(* CODESYS project barrier.v1.12.paramReset.project

Project tree, tasks and I/O mapping:
  Device : ShenZhen RenTong SoftMotion RTE V3,  Shenzhen Rentong IST LTD, order no. 309015, version 3.5.9.50
    application Application
      libraries: Standard, * (System); VisuDialogs, * (System); SysDir, 3.5.8.0 (System); SysTime23, 3.5.2.0 (System); TCP, 3.5.9.50 (3S - Smart Software Solutions GmbH); SysFile, 3.5.9.0 (System); SysStr23, 3.5.8.0 (System); modbus tcp serverAndClient, 1.0.1 (深圳人通长沙研究院); ModbusTCP Slave, 3.5.10.0 (3S - Smart Software Solutions GmbH)
      task CAN_TX (cyclic, interval t#10ms, priority 1) calls CanTx
      task CAN_RX (cyclic, interval 6 ms, priority 1) calls CanRx
      task MAIN (cyclic, interval t#10ms, priority 2) calls Barrier
      task VISU_TASK (cyclic, interval 100 ms, priority 31) calls VisuElems.Visu_Prg
      task MODBUS (cyclic, interval t#10ms, priority 1) calls ModbusAct
      task ETHERCAT (cyclic, interval 2000 µs, priority 0) calls EtherCAT_Master.EtherCAT_Task [EtherCAT_Master.EtherCAT_Task]
      task HEALTHY_DATA1 (cyclic, interval t#500ms, priority 1) calls TcpUploader
      task HEALTHY_DATA2 (cyclic, interval t#10ms, priority 1) calls FileSaver
      basestruct/
        data type CmdPercentSet
        data type SensorInfo
        data type DeviceUnit
        data type UIMode
        data type UIUnit
        data type TargetDirect
        data type DevStatus
      can/
        canstruct/
          data type Can_BUS_8Inputs
          data type Can_BUS_8Outputs
          data type Can_Bus_RXMsg_Buff
          data type Can_Bus_TXMsg_Buff
          data type Can_baseframe
        program CanTx [ST]: C01_Tx, C02_Tx, C03_Tx, C04_Tx, C05_Tx, C06_Tx
        program CanRx [ST]: C01_Rx, C02_Rx, C03_Rx, C04_Rx, C05_Rx, C06_Rx
        function CAN_Read_Data_SWMC [ST]
        function CAN_Send_Data_SWMC [ST]
      global/
        global variables gController
        global variables gCan
        global variables gDev
        global variables gUI
        global variables gModbus
      visualization/
        baseModule/
          visualisation DevUnit0
          visualisation grd
          visualisation setting
          visualisation sky
          visualisation BasePID
          visualisation testPID
          visualisation currentUnit
      core/
        program Barrier [ST]: updateStatus, initialize, interfaceAct, autoResetButton, manualExecute, pidExecute, pidTestUi, autoEnable, pidCalc, setExecutePercent, initializePid
        pid/
          function block BasePIDCtrl [ST]
          data type PidParam
          data type UiPid
          data type DevPid
          function block grdPosCtrl [ST]
          function block skyPosCtrl [ST]
          data type FeedForward
      visualisation main
      healthydata/
        program TcpUploader [ST]: prepareMetaData
        program FileSaver [ST]: getSkyData, getGrdData
      modbus/
        struct/
          data type mdbsStruct
          data type mdbsRequest
          data type mdbsResponse
        program ModbusAct [ST]: initialize, localCmdHandler, updateStat, handleCmd, handleStat1, handleStat2, handleStat3, localStatHandler
        function block mdbsLogicToPhy [ST]
        function block mdbsPhyToLogic [ST]
        function block mdbsNumToIdx [ST]
        function block DataReverse [ST]: cmdReverse
      atrace/
        trace delay_g_07 (task MAIN, trigger Positive on CanRx.count 1): gController.grd[7].retractPercent, gController.grd[7].extendPercent, gDev.grd[7].sensor.position, gDev.grd[7].sensor.speed
        trace show (task MAIN, trigger Positive on CanRx.count 1): gDev.grd[9].sensor.position, gDev.grd[9].sensor.speed, Barrier.grdPid[9].res, gController.grd[9].retractPercent, gController.grd[9].extendPercent, gDev.sky[9].sensor.position, gDev.sky[9].sensor.speed, Barrier.skyPid[9].res, gController.sky[9].retractPercent, gController.sky[9].extendPercent
        trace delay_g_08 (task MAIN, trigger Positive on CanRx.count 1): gController.grd[8].retractPercent, gController.grd[8].extendPercent, gDev.grd[8].sensor.position, gDev.grd[8].sensor.speed
        trace show2 (task MAIN, trigger Positive on CanRx.count 1): gController.grd[1].retractPercent, gController.grd[1].extendPercent, gDev.grd[1].sensor.position, gDev.grd[1].sensor.speed
        sync/
          trace delay_sync_01 (task MAIN, trigger Positive on CanRx.count 1): gDev.grd[1].sensor.position, gDev.grd[1].sensor.speed, gDev.sky[1].sensor.position, gDev.sky[1].sensor.speed
          trace delay_sync_02 (task MAIN, trigger Positive on CanRx.count 1): gDev.grd[2].sensor.position, gDev.grd[2].sensor.speed, gDev.sky[2].sensor.position, gDev.sky[2].sensor.speed
          trace delay_sync_03 (task MAIN, trigger Positive on CanRx.count 1): gDev.grd[3].sensor.position, gDev.grd[3].sensor.speed, gDev.sky[3].sensor.position, gDev.sky[3].sensor.speed
          trace delay_sync_04 (task MAIN, trigger Positive on CanRx.count 1): gDev.grd[4].sensor.position, gDev.grd[4].sensor.speed, gDev.sky[4].sensor.position, gDev.sky[4].sensor.speed
          trace delay_sync_05 (task MAIN, trigger Positive on CanRx.count 1): gDev.grd[5].sensor.position, gDev.grd[5].sensor.speed, gDev.sky[5].sensor.position, gDev.sky[5].sensor.speed
          trace delay_sync_06 (task MAIN, trigger Positive on CanRx.count 1): gDev.grd[6].sensor.position, gDev.grd[6].sensor.speed, gDev.sky[6].sensor.position, gDev.sky[6].sensor.speed
          trace delay_sync_07 (task MAIN, trigger Positive on CanRx.count 1): gDev.grd[7].sensor.position, gDev.grd[7].sensor.speed, gDev.sky[7].sensor.position, gDev.sky[7].sensor.speed
          trace delay_sync_08 (task MAIN, trigger Positive on CanRx.count 1): gDev.grd[8].sensor.position, gDev.grd[8].sensor.speed, gDev.sky[8].sensor.position, gDev.sky[8].sensor.speed
          trace delay_sync_09 (task MAIN, trigger Positive on CanRx.count 1): gDev.grd[9].sensor.position, gDev.grd[9].sensor.speed, gDev.sky[9].sensor.position, gDev.sky[9].sensor.speed
          trace delay_sync_10 (task MAIN, trigger Positive on CanRx.count 1): gDev.grd[10].sensor.position, gDev.grd[10].sensor.speed, gDev.sky[10].sensor.position, gDev.sky[10].sensor.speed
        last/
          trace delay_s_0 (task MAIN, trigger Positive on CanRx.count 1): gController.sky[0].retractPercent, gController.sky[0].extendPercent, gDev.sky[0].sensor.position, gDev.sky[0].sensor.speed
          trace delay_g_5 (task MAIN, trigger Positive on CanRx.count 1): gController.grd[5].retractPercent, gController.grd[5].extendPercent, gDev.grd[5].sensor.position, gDev.grd[5].sensor.speed
          trace delay_g_1 (task MAIN, trigger Positive on CanRx.count 1): gController.grd[1].retractPercent, gController.grd[1].extendPercent, gDev.grd[1].sensor.position, gDev.grd[1].sensor.speed
          trace delay_g_2 (task MAIN, trigger Positive on CanRx.count 1): gController.grd[2].retractPercent, gController.grd[2].extendPercent, gDev.grd[2].sensor.position, gDev.grd[2].sensor.speed
          trace delay_g_3 (task MAIN, trigger Positive on CanRx.count 1): gController.grd[3].retractPercent, gController.grd[3].extendPercent, gDev.grd[3].current[1], gDev.grd[3].current[2], gDev.grd[3].sensor.position, gDev.grd[3].sensor.speed
          trace delay_g_4 (task MAIN, trigger Positive on CanRx.count 1): gController.grd[4].retractPercent, gController.grd[4].extendPercent, gDev.grd[4].current[1], gDev.grd[4].current[2], gDev.grd[4].sensor.position, gDev.grd[4].sensor.speed
          trace delay_g_6 (task MAIN, trigger Positive on CanRx.count 1): gController.grd[6].retractPercent, gController.grd[6].extendPercent, gDev.grd[6].current[1], gDev.grd[6].current[2], gDev.grd[6].sensor.position, gDev.grd[6].sensor.speed
          trace delay_s_6 (task MAIN, trigger Positive on CanRx.count 1): gController.sky[6].retractPercent, gController.sky[6].extendPercent, gDev.sky[6].sensor.position, gDev.sky[6].sensor.speed
          trace delay_s_5 (task MAIN, trigger Positive on CanRx.count 1): gController.sky[5].retractPercent, gController.sky[5].extendPercent, gDev.sky[5].sensor.position, gDev.sky[5].sensor.speed
          trace delay_s_4 (task MAIN, trigger Positive on CanRx.count 1): gController.sky[4].retractPercent, gController.sky[4].extendPercent, gDev.sky[4].sensor.position, gDev.sky[4].sensor.speed
          trace delay_s_3 (task MAIN, trigger Positive on CanRx.count 1): gController.sky[3].retractPercent, gController.sky[3].extendPercent, gDev.sky[3].sensor.position, gDev.sky[3].sensor.speed
          trace delay_s_2 (task MAIN, trigger Positive on CanRx.count 1): gController.sky[2].retractPercent, gController.sky[2].extendPercent, gDev.sky[2].sensor.position, gDev.sky[2].sensor.speed
          trace delay_s_1 (task MAIN, trigger Positive on CanRx.count 1): gController.sky[1].retractPercent, gController.sky[1].extendPercent, gDev.sky[1].sensor.position, gDev.sky[1].sensor.speed
        trace delay_g_09 (task MAIN, trigger Positive on CanRx.count 1): gController.grd[9].retractPercent, gController.grd[9].extendPercent, gDev.grd[9].sensor.position, gDev.grd[9].sensor.speed
        trace delay_g_10 (task MAIN, trigger Positive on CanRx.count 1): gController.grd[10].retractPercent, gController.grd[10].extendPercent, gDev.grd[10].sensor.position, gDev.grd[10].sensor.speed
        trace delay_s_07 (task MAIN, trigger Positive on CanRx.count 1): gController.sky[07].retractPercent, gController.sky[07].extendPercent, gDev.sky[07].sensor.position, gDev.sky[07].sensor.speed
        trace delay_s_08 (task MAIN, trigger Positive on CanRx.count 1): gController.sky[8].retractPercent, gController.sky[8].extendPercent, gDev.sky[8].sensor.position, gDev.sky[8].sensor.speed
        trace delay_s_09 (task MAIN, trigger Positive on CanRx.count 1): gDev.grd[9].sensor.position, gDev.grd[9].sensor.speed, Barrier.grdPid[9].res, gController.grd[9].retractPercent, gController.grd[9].extendPercent, gDev.sky[9].sensor.position, gDev.sky[9].sensor.speed, Barrier.skyPid[9].res, gController.sky[9].retractPercent, gController.sky[9].extendPercent
        trace delay_s_10 (task MAIN, trigger Positive on CanRx.count 1): gController.sky[10].retractPercent, gController.sky[10].extendPercent, gDev.sky[10].sensor.position, gDev.sky[10].sensor.speed
      basefun/
        function block CommandExecutor0 [ST]
        function percentCalc [ST]
        function setButtonByDirect [ST]
        function updateDevStatus [ST]
        function block tcpUpload [ST]: send
        function block fileSave [ST]: new, close, write, createDir
        function block CommandExecutor [ST]
    SoftMotion General Axis Pool
    EtherCAT_Master : EtherCAT Master, 3S - Smart Software Solutions GmbH, version 3.5.10.0
        settings: MasterCycleTime = 2000; NetworkName = '本地连接 5'; NetworkName = "本地连接 5"; SrcAddress1 = 26861; SrcAddress2 = 2754393510
      EK1100_0030 : EK1100-0030 EtherCAT Coupler (2A E-Bus, 4kV galv. iso.), Beckhoff Automation GmbH & Co. KG, order no. EK1100-0030, version Revision=16#0011001E
          settings: DC sync0 cycletime = 2000; DC sync1 cycletime = 2000
        EL6751_CANMiniDriver : EL6751 CAN MiniDriver (8 Messages), Beckhoff Automation GmbH, version 3.5.9.0
            settings: DC sync0 cycletime = 2000; DC sync1 cycletime = 2000
            unmapped channels: TxCounter, RxCounter, NoOfTxMessages, TxMsg1_TransactionNumber, TxMsg1_CobId, TxMsg1_Byte1, TxMsg1_Byte2, TxMsg1_Byte3, TxMsg1_Byte4, TxMsg1_Byte5, TxMsg1_Byte6, TxMsg1_Byte7, TxMsg1_Byte8, TxMsg2_TransactionNumber, TxMsg2_CobId, TxMsg2_Byte1, TxMsg2_Byte2, TxMsg2_Byte3, TxMsg2_Byte4, TxMsg2_Byte5, TxMsg2_Byte6, TxMsg2_Byte7, TxMsg2_Byte8, TxMsg3_TransactionNumber, TxMsg3_CobId, TxMsg3_Byte1, TxMsg3_Byte2, TxMsg3_Byte3, TxMsg3_Byte4, TxMsg3_Byte5, TxMsg3_Byte6, TxMsg3_Byte7, TxMsg3_Byte8, TxMsg4_TransactionNumber, TxMsg4_CobId, TxMsg4_Byte1, TxMsg4_Byte2, TxMsg4_Byte3, TxMsg4_Byte4, TxMsg4_Byte5,
              TxMsg4_Byte6, TxMsg4_Byte7, TxMsg4_Byte8, TxMsg5_TransactionNumber, TxMsg5_CobId, TxMsg5_Byte1, TxMsg5_Byte2, TxMsg5_Byte3, TxMsg5_Byte4, TxMsg5_Byte5, TxMsg5_Byte6, TxMsg5_Byte7, TxMsg5_Byte8, TxMsg6_TransactionNumber, TxMsg6_CobId, TxMsg6_Byte1, TxMsg6_Byte2, TxMsg6_Byte3, TxMsg6_Byte4, TxMsg6_Byte5, TxMsg6_Byte6, TxMsg6_Byte7, TxMsg6_Byte8, TxMsg7_TransactionNumber, TxMsg7_CobId, TxMsg7_Byte1, TxMsg7_Byte2, TxMsg7_Byte3, TxMsg7_Byte4, TxMsg7_Byte5, TxMsg7_Byte6, TxMsg7_Byte7, TxMsg7_Byte8, TxMsg8_TransactionNumber, TxMsg8_CobId, TxMsg8_Byte1, TxMsg8_Byte2, TxMsg8_Byte3, TxMsg8_Byte4, TxMsg8_Byte5,
              TxMsg8_Byte6, TxMsg8_Byte7, TxMsg8_Byte8, CAN Control, TxCounter, RxCounter, NoOfRxMessages, TransactionNumber, RxMsg1_CobId, RxMsg1_Byte1, RxMsg1_Byte2, RxMsg1_Byte3, RxMsg1_Byte4, RxMsg1_Byte5, RxMsg1_Byte6, RxMsg1_Byte7, RxMsg1_Byte8, RxMsg2_CobId, RxMsg2_Byte1, RxMsg2_Byte2, RxMsg2_Byte3, RxMsg2_Byte4, RxMsg2_Byte5, RxMsg2_Byte6, RxMsg2_Byte7, RxMsg2_Byte8, RxMsg3_CobId, RxMsg3_Byte1, RxMsg3_Byte2, RxMsg3_Byte3, RxMsg3_Byte4, RxMsg3_Byte5, RxMsg3_Byte6, RxMsg3_Byte7, RxMsg3_Byte8, RxMsg4_CobId, RxMsg4_Byte1, RxMsg4_Byte2, RxMsg4_Byte3, RxMsg4_Byte4,
              RxMsg4_Byte5, RxMsg4_Byte6, RxMsg4_Byte7, RxMsg4_Byte8, RxMsg5_CobId, RxMsg5_Byte1, RxMsg5_Byte2, RxMsg5_Byte3, RxMsg5_Byte4, RxMsg5_Byte5, RxMsg5_Byte6, RxMsg5_Byte7, RxMsg5_Byte8, RxMsg6_CobId, RxMsg6_Byte1, RxMsg6_Byte2, RxMsg6_Byte3, RxMsg6_Byte4, RxMsg6_Byte5, RxMsg6_Byte6, RxMsg6_Byte7, RxMsg6_Byte8, RxMsg7_CobId, RxMsg7_Byte1, RxMsg7_Byte2, RxMsg7_Byte3, RxMsg7_Byte4, RxMsg7_Byte5, RxMsg7_Byte6, RxMsg7_Byte7, RxMsg7_Byte8, RxMsg8_CobId, RxMsg8_Byte1, RxMsg8_Byte2, RxMsg8_Byte3, RxMsg8_Byte4, RxMsg8_Byte5, RxMsg8_Byte6, RxMsg8_Byte7, RxMsg8_Byte8,
              CAN State, Align, RX Error Counter, TX Error Counter
          CANbus
      EK1100_0030_1 : EK1100-0030 EtherCAT Coupler (2A E-Bus, 4kV galv. iso.), Beckhoff Automation GmbH & Co. KG, order no. EK1100-0030, version Revision=16#0011001E
          settings: DC sync0 cycletime = 2000; DC sync1 cycletime = 2000
        EL6751_CANMiniDriver_1 : EL6751 CAN MiniDriver (8 Messages), Beckhoff Automation GmbH, version 3.5.9.0
            settings: DC sync0 cycletime = 2000; DC sync1 cycletime = 2000
            unmapped channels: TxCounter, RxCounter, NoOfTxMessages, TxMsg1_TransactionNumber, TxMsg1_CobId, TxMsg1_Byte1, TxMsg1_Byte2, TxMsg1_Byte3, TxMsg1_Byte4, TxMsg1_Byte5, TxMsg1_Byte6, TxMsg1_Byte7, TxMsg1_Byte8, TxMsg2_TransactionNumber, TxMsg2_CobId, TxMsg2_Byte1, TxMsg2_Byte2, TxMsg2_Byte3, TxMsg2_Byte4, TxMsg2_Byte5, TxMsg2_Byte6, TxMsg2_Byte7, TxMsg2_Byte8, TxMsg3_TransactionNumber, TxMsg3_CobId, TxMsg3_Byte1, TxMsg3_Byte2, TxMsg3_Byte3, TxMsg3_Byte4, TxMsg3_Byte5, TxMsg3_Byte6, TxMsg3_Byte7, TxMsg3_Byte8, TxMsg4_TransactionNumber, TxMsg4_CobId, TxMsg4_Byte1, TxMsg4_Byte2, TxMsg4_Byte3, TxMsg4_Byte4, TxMsg4_Byte5,
              TxMsg4_Byte6, TxMsg4_Byte7, TxMsg4_Byte8, TxMsg5_TransactionNumber, TxMsg5_CobId, TxMsg5_Byte1, TxMsg5_Byte2, TxMsg5_Byte3, TxMsg5_Byte4, TxMsg5_Byte5, TxMsg5_Byte6, TxMsg5_Byte7, TxMsg5_Byte8, TxMsg6_TransactionNumber, TxMsg6_CobId, TxMsg6_Byte1, TxMsg6_Byte2, TxMsg6_Byte3, TxMsg6_Byte4, TxMsg6_Byte5, TxMsg6_Byte6, TxMsg6_Byte7, TxMsg6_Byte8, TxMsg7_TransactionNumber, TxMsg7_CobId, TxMsg7_Byte1, TxMsg7_Byte2, TxMsg7_Byte3, TxMsg7_Byte4, TxMsg7_Byte5, TxMsg7_Byte6, TxMsg7_Byte7, TxMsg7_Byte8, TxMsg8_TransactionNumber, TxMsg8_CobId, TxMsg8_Byte1, TxMsg8_Byte2, TxMsg8_Byte3, TxMsg8_Byte4, TxMsg8_Byte5,
              TxMsg8_Byte6, TxMsg8_Byte7, TxMsg8_Byte8, CAN Control, TxCounter, RxCounter, NoOfRxMessages, TransactionNumber, RxMsg1_CobId, RxMsg1_Byte1, RxMsg1_Byte2, RxMsg1_Byte3, RxMsg1_Byte4, RxMsg1_Byte5, RxMsg1_Byte6, RxMsg1_Byte7, RxMsg1_Byte8, RxMsg2_CobId, RxMsg2_Byte1, RxMsg2_Byte2, RxMsg2_Byte3, RxMsg2_Byte4, RxMsg2_Byte5, RxMsg2_Byte6, RxMsg2_Byte7, RxMsg2_Byte8, RxMsg3_CobId, RxMsg3_Byte1, RxMsg3_Byte2, RxMsg3_Byte3, RxMsg3_Byte4, RxMsg3_Byte5, RxMsg3_Byte6, RxMsg3_Byte7, RxMsg3_Byte8, RxMsg4_CobId, RxMsg4_Byte1, RxMsg4_Byte2, RxMsg4_Byte3, RxMsg4_Byte4,
              RxMsg4_Byte5, RxMsg4_Byte6, RxMsg4_Byte7, RxMsg4_Byte8, RxMsg5_CobId, RxMsg5_Byte1, RxMsg5_Byte2, RxMsg5_Byte3, RxMsg5_Byte4, RxMsg5_Byte5, RxMsg5_Byte6, RxMsg5_Byte7, RxMsg5_Byte8, RxMsg6_CobId, RxMsg6_Byte1, RxMsg6_Byte2, RxMsg6_Byte3, RxMsg6_Byte4, RxMsg6_Byte5, RxMsg6_Byte6, RxMsg6_Byte7, RxMsg6_Byte8, RxMsg7_CobId, RxMsg7_Byte1, RxMsg7_Byte2, RxMsg7_Byte3, RxMsg7_Byte4, RxMsg7_Byte5, RxMsg7_Byte6, RxMsg7_Byte7, RxMsg7_Byte8, RxMsg8_CobId, RxMsg8_Byte1, RxMsg8_Byte2, RxMsg8_Byte3, RxMsg8_Byte4, RxMsg8_Byte5, RxMsg8_Byte6, RxMsg8_Byte7, RxMsg8_Byte8,
              CAN State, Align, RX Error Counter, TX Error Counter
          CANbus
              settings: NetID = 1
      EK1100_0030_2 : EK1100-0030 EtherCAT Coupler (2A E-Bus, 4kV galv. iso.), Beckhoff Automation GmbH & Co. KG, order no. EK1100-0030, version Revision=16#0011001E
          settings: DC sync0 cycletime = 2000; DC sync1 cycletime = 2000
        EL6751_CANMiniDriver_2 : EL6751 CAN MiniDriver (8 Messages), Beckhoff Automation GmbH, version 3.5.9.0
            settings: DC sync0 cycletime = 2000; DC sync1 cycletime = 2000
            unmapped channels: TxCounter, RxCounter, NoOfTxMessages, TxMsg1_TransactionNumber, TxMsg1_CobId, TxMsg1_Byte1, TxMsg1_Byte2, TxMsg1_Byte3, TxMsg1_Byte4, TxMsg1_Byte5, TxMsg1_Byte6, TxMsg1_Byte7, TxMsg1_Byte8, TxMsg2_TransactionNumber, TxMsg2_CobId, TxMsg2_Byte1, TxMsg2_Byte2, TxMsg2_Byte3, TxMsg2_Byte4, TxMsg2_Byte5, TxMsg2_Byte6, TxMsg2_Byte7, TxMsg2_Byte8, TxMsg3_TransactionNumber, TxMsg3_CobId, TxMsg3_Byte1, TxMsg3_Byte2, TxMsg3_Byte3, TxMsg3_Byte4, TxMsg3_Byte5, TxMsg3_Byte6, TxMsg3_Byte7, TxMsg3_Byte8, TxMsg4_TransactionNumber, TxMsg4_CobId, TxMsg4_Byte1, TxMsg4_Byte2, TxMsg4_Byte3, TxMsg4_Byte4, TxMsg4_Byte5,
              TxMsg4_Byte6, TxMsg4_Byte7, TxMsg4_Byte8, TxMsg5_TransactionNumber, TxMsg5_CobId, TxMsg5_Byte1, TxMsg5_Byte2, TxMsg5_Byte3, TxMsg5_Byte4, TxMsg5_Byte5, TxMsg5_Byte6, TxMsg5_Byte7, TxMsg5_Byte8, TxMsg6_TransactionNumber, TxMsg6_CobId, TxMsg6_Byte1, TxMsg6_Byte2, TxMsg6_Byte3, TxMsg6_Byte4, TxMsg6_Byte5, TxMsg6_Byte6, TxMsg6_Byte7, TxMsg6_Byte8, TxMsg7_TransactionNumber, TxMsg7_CobId, TxMsg7_Byte1, TxMsg7_Byte2, TxMsg7_Byte3, TxMsg7_Byte4, TxMsg7_Byte5, TxMsg7_Byte6, TxMsg7_Byte7, TxMsg7_Byte8, TxMsg8_TransactionNumber, TxMsg8_CobId, TxMsg8_Byte1, TxMsg8_Byte2, TxMsg8_Byte3, TxMsg8_Byte4, TxMsg8_Byte5,
              TxMsg8_Byte6, TxMsg8_Byte7, TxMsg8_Byte8, CAN Control, TxCounter, RxCounter, NoOfRxMessages, TransactionNumber, RxMsg1_CobId, RxMsg1_Byte1, RxMsg1_Byte2, RxMsg1_Byte3, RxMsg1_Byte4, RxMsg1_Byte5, RxMsg1_Byte6, RxMsg1_Byte7, RxMsg1_Byte8, RxMsg2_CobId, RxMsg2_Byte1, RxMsg2_Byte2, RxMsg2_Byte3, RxMsg2_Byte4, RxMsg2_Byte5, RxMsg2_Byte6, RxMsg2_Byte7, RxMsg2_Byte8, RxMsg3_CobId, RxMsg3_Byte1, RxMsg3_Byte2, RxMsg3_Byte3, RxMsg3_Byte4, RxMsg3_Byte5, RxMsg3_Byte6, RxMsg3_Byte7, RxMsg3_Byte8, RxMsg4_CobId, RxMsg4_Byte1, RxMsg4_Byte2, RxMsg4_Byte3, RxMsg4_Byte4,
              RxMsg4_Byte5, RxMsg4_Byte6, RxMsg4_Byte7, RxMsg4_Byte8, RxMsg5_CobId, RxMsg5_Byte1, RxMsg5_Byte2, RxMsg5_Byte3, RxMsg5_Byte4, RxMsg5_Byte5, RxMsg5_Byte6, RxMsg5_Byte7, RxMsg5_Byte8, RxMsg6_CobId, RxMsg6_Byte1, RxMsg6_Byte2, RxMsg6_Byte3, RxMsg6_Byte4, RxMsg6_Byte5, RxMsg6_Byte6, RxMsg6_Byte7, RxMsg6_Byte8, RxMsg7_CobId, RxMsg7_Byte1, RxMsg7_Byte2, RxMsg7_Byte3, RxMsg7_Byte4, RxMsg7_Byte5, RxMsg7_Byte6, RxMsg7_Byte7, RxMsg7_Byte8, RxMsg8_CobId, RxMsg8_Byte1, RxMsg8_Byte2, RxMsg8_Byte3, RxMsg8_Byte4, RxMsg8_Byte5, RxMsg8_Byte6, RxMsg8_Byte7, RxMsg8_Byte8,
              CAN State, Align, RX Error Counter, TX Error Counter
          CANbus
              settings: NetID = 2
      EK1100_0030_3 : EK1100-0030 EtherCAT Coupler (2A E-Bus, 4kV galv. iso.), Beckhoff Automation GmbH & Co. KG, order no. EK1100-0030, version Revision=16#0011001E
          settings: DC sync0 cycletime = 2000; DC sync1 cycletime = 2000
        EL6751_CANMiniDriver_3 : EL6751 CAN MiniDriver (8 Messages), Beckhoff Automation GmbH, version 3.5.9.0
            settings: DC sync0 cycletime = 2000; DC sync1 cycletime = 2000
            unmapped channels: TxCounter, RxCounter, NoOfTxMessages, TxMsg1_TransactionNumber, TxMsg1_CobId, TxMsg1_Byte1, TxMsg1_Byte2, TxMsg1_Byte3, TxMsg1_Byte4, TxMsg1_Byte5, TxMsg1_Byte6, TxMsg1_Byte7, TxMsg1_Byte8, TxMsg2_TransactionNumber, TxMsg2_CobId, TxMsg2_Byte1, TxMsg2_Byte2, TxMsg2_Byte3, TxMsg2_Byte4, TxMsg2_Byte5, TxMsg2_Byte6, TxMsg2_Byte7, TxMsg2_Byte8, TxMsg3_TransactionNumber, TxMsg3_CobId, TxMsg3_Byte1, TxMsg3_Byte2, TxMsg3_Byte3, TxMsg3_Byte4, TxMsg3_Byte5, TxMsg3_Byte6, TxMsg3_Byte7, TxMsg3_Byte8, TxMsg4_TransactionNumber, TxMsg4_CobId, TxMsg4_Byte1, TxMsg4_Byte2, TxMsg4_Byte3, TxMsg4_Byte4, TxMsg4_Byte5,
              TxMsg4_Byte6, TxMsg4_Byte7, TxMsg4_Byte8, TxMsg5_TransactionNumber, TxMsg5_CobId, TxMsg5_Byte1, TxMsg5_Byte2, TxMsg5_Byte3, TxMsg5_Byte4, TxMsg5_Byte5, TxMsg5_Byte6, TxMsg5_Byte7, TxMsg5_Byte8, TxMsg6_TransactionNumber, TxMsg6_CobId, TxMsg6_Byte1, TxMsg6_Byte2, TxMsg6_Byte3, TxMsg6_Byte4, TxMsg6_Byte5, TxMsg6_Byte6, TxMsg6_Byte7, TxMsg6_Byte8, TxMsg7_TransactionNumber, TxMsg7_CobId, TxMsg7_Byte1, TxMsg7_Byte2, TxMsg7_Byte3, TxMsg7_Byte4, TxMsg7_Byte5, TxMsg7_Byte6, TxMsg7_Byte7, TxMsg7_Byte8, TxMsg8_TransactionNumber, TxMsg8_CobId, TxMsg8_Byte1, TxMsg8_Byte2, TxMsg8_Byte3, TxMsg8_Byte4, TxMsg8_Byte5,
              TxMsg8_Byte6, TxMsg8_Byte7, TxMsg8_Byte8, CAN Control, TxCounter, RxCounter, NoOfRxMessages, TransactionNumber, RxMsg1_CobId, RxMsg1_Byte1, RxMsg1_Byte2, RxMsg1_Byte3, RxMsg1_Byte4, RxMsg1_Byte5, RxMsg1_Byte6, RxMsg1_Byte7, RxMsg1_Byte8, RxMsg2_CobId, RxMsg2_Byte1, RxMsg2_Byte2, RxMsg2_Byte3, RxMsg2_Byte4, RxMsg2_Byte5, RxMsg2_Byte6, RxMsg2_Byte7, RxMsg2_Byte8, RxMsg3_CobId, RxMsg3_Byte1, RxMsg3_Byte2, RxMsg3_Byte3, RxMsg3_Byte4, RxMsg3_Byte5, RxMsg3_Byte6, RxMsg3_Byte7, RxMsg3_Byte8, RxMsg4_CobId, RxMsg4_Byte1, RxMsg4_Byte2, RxMsg4_Byte3, RxMsg4_Byte4,
              RxMsg4_Byte5, RxMsg4_Byte6, RxMsg4_Byte7, RxMsg4_Byte8, RxMsg5_CobId, RxMsg5_Byte1, RxMsg5_Byte2, RxMsg5_Byte3, RxMsg5_Byte4, RxMsg5_Byte5, RxMsg5_Byte6, RxMsg5_Byte7, RxMsg5_Byte8, RxMsg6_CobId, RxMsg6_Byte1, RxMsg6_Byte2, RxMsg6_Byte3, RxMsg6_Byte4, RxMsg6_Byte5, RxMsg6_Byte6, RxMsg6_Byte7, RxMsg6_Byte8, RxMsg7_CobId, RxMsg7_Byte1, RxMsg7_Byte2, RxMsg7_Byte3, RxMsg7_Byte4, RxMsg7_Byte5, RxMsg7_Byte6, RxMsg7_Byte7, RxMsg7_Byte8, RxMsg8_CobId, RxMsg8_Byte1, RxMsg8_Byte2, RxMsg8_Byte3, RxMsg8_Byte4, RxMsg8_Byte5, RxMsg8_Byte6, RxMsg8_Byte7, RxMsg8_Byte8,
              CAN State, Align, RX Error Counter, TX Error Counter
          CANbus
              settings: NetID = 3
      EK1100_0030_4 : EK1100-0030 EtherCAT Coupler (2A E-Bus, 4kV galv. iso.), Beckhoff Automation GmbH & Co. KG, order no. EK1100-0030, version Revision=16#0011001E
          settings: DC sync0 cycletime = 2000; DC sync1 cycletime = 2000
        EL6751_CANMiniDriver_4 : EL6751 CAN MiniDriver (8 Messages), Beckhoff Automation GmbH, version 3.5.9.0
            settings: DC sync0 cycletime = 2000; DC sync1 cycletime = 2000
            unmapped channels: TxCounter, RxCounter, NoOfTxMessages, TxMsg1_TransactionNumber, TxMsg1_CobId, TxMsg1_Byte1, TxMsg1_Byte2, TxMsg1_Byte3, TxMsg1_Byte4, TxMsg1_Byte5, TxMsg1_Byte6, TxMsg1_Byte7, TxMsg1_Byte8, TxMsg2_TransactionNumber, TxMsg2_CobId, TxMsg2_Byte1, TxMsg2_Byte2, TxMsg2_Byte3, TxMsg2_Byte4, TxMsg2_Byte5, TxMsg2_Byte6, TxMsg2_Byte7, TxMsg2_Byte8, TxMsg3_TransactionNumber, TxMsg3_CobId, TxMsg3_Byte1, TxMsg3_Byte2, TxMsg3_Byte3, TxMsg3_Byte4, TxMsg3_Byte5, TxMsg3_Byte6, TxMsg3_Byte7, TxMsg3_Byte8, TxMsg4_TransactionNumber, TxMsg4_CobId, TxMsg4_Byte1, TxMsg4_Byte2, TxMsg4_Byte3, TxMsg4_Byte4, TxMsg4_Byte5,
              TxMsg4_Byte6, TxMsg4_Byte7, TxMsg4_Byte8, TxMsg5_TransactionNumber, TxMsg5_CobId, TxMsg5_Byte1, TxMsg5_Byte2, TxMsg5_Byte3, TxMsg5_Byte4, TxMsg5_Byte5, TxMsg5_Byte6, TxMsg5_Byte7, TxMsg5_Byte8, TxMsg6_TransactionNumber, TxMsg6_CobId, TxMsg6_Byte1, TxMsg6_Byte2, TxMsg6_Byte3, TxMsg6_Byte4, TxMsg6_Byte5, TxMsg6_Byte6, TxMsg6_Byte7, TxMsg6_Byte8, TxMsg7_TransactionNumber, TxMsg7_CobId, TxMsg7_Byte1, TxMsg7_Byte2, TxMsg7_Byte3, TxMsg7_Byte4, TxMsg7_Byte5, TxMsg7_Byte6, TxMsg7_Byte7, TxMsg7_Byte8, TxMsg8_TransactionNumber, TxMsg8_CobId, TxMsg8_Byte1, TxMsg8_Byte2, TxMsg8_Byte3, TxMsg8_Byte4, TxMsg8_Byte5,
              TxMsg8_Byte6, TxMsg8_Byte7, TxMsg8_Byte8, CAN Control, TxCounter, RxCounter, NoOfRxMessages, TransactionNumber, RxMsg1_CobId, RxMsg1_Byte1, RxMsg1_Byte2, RxMsg1_Byte3, RxMsg1_Byte4, RxMsg1_Byte5, RxMsg1_Byte6, RxMsg1_Byte7, RxMsg1_Byte8, RxMsg2_CobId, RxMsg2_Byte1, RxMsg2_Byte2, RxMsg2_Byte3, RxMsg2_Byte4, RxMsg2_Byte5, RxMsg2_Byte6, RxMsg2_Byte7, RxMsg2_Byte8, RxMsg3_CobId, RxMsg3_Byte1, RxMsg3_Byte2, RxMsg3_Byte3, RxMsg3_Byte4, RxMsg3_Byte5, RxMsg3_Byte6, RxMsg3_Byte7, RxMsg3_Byte8, RxMsg4_CobId, RxMsg4_Byte1, RxMsg4_Byte2, RxMsg4_Byte3, RxMsg4_Byte4,
              RxMsg4_Byte5, RxMsg4_Byte6, RxMsg4_Byte7, RxMsg4_Byte8, RxMsg5_CobId, RxMsg5_Byte1, RxMsg5_Byte2, RxMsg5_Byte3, RxMsg5_Byte4, RxMsg5_Byte5, RxMsg5_Byte6, RxMsg5_Byte7, RxMsg5_Byte8, RxMsg6_CobId, RxMsg6_Byte1, RxMsg6_Byte2, RxMsg6_Byte3, RxMsg6_Byte4, RxMsg6_Byte5, RxMsg6_Byte6, RxMsg6_Byte7, RxMsg6_Byte8, RxMsg7_CobId, RxMsg7_Byte1, RxMsg7_Byte2, RxMsg7_Byte3, RxMsg7_Byte4, RxMsg7_Byte5, RxMsg7_Byte6, RxMsg7_Byte7, RxMsg7_Byte8, RxMsg8_CobId, RxMsg8_Byte1, RxMsg8_Byte2, RxMsg8_Byte3, RxMsg8_Byte4, RxMsg8_Byte5, RxMsg8_Byte6, RxMsg8_Byte7, RxMsg8_Byte8,
              CAN State, Align, RX Error Counter, TX Error Counter
          CANbus
              settings: NetID = 4
      EK1100_0030_5 : EK1100-0030 EtherCAT Coupler (2A E-Bus, 4kV galv. iso.), Beckhoff Automation GmbH & Co. KG, order no. EK1100-0030, version Revision=16#0011001E
          settings: DC sync0 cycletime = 2000; DC sync1 cycletime = 2000
        EL6751_CANMiniDriver_5 : EL6751 CAN MiniDriver (8 Messages), Beckhoff Automation GmbH, version 3.5.9.0
            settings: DC sync0 cycletime = 2000; DC sync1 cycletime = 2000
            unmapped channels: TxCounter, RxCounter, NoOfTxMessages, TxMsg1_TransactionNumber, TxMsg1_CobId, TxMsg1_Byte1, TxMsg1_Byte2, TxMsg1_Byte3, TxMsg1_Byte4, TxMsg1_Byte5, TxMsg1_Byte6, TxMsg1_Byte7, TxMsg1_Byte8, TxMsg2_TransactionNumber, TxMsg2_CobId, TxMsg2_Byte1, TxMsg2_Byte2, TxMsg2_Byte3, TxMsg2_Byte4, TxMsg2_Byte5, TxMsg2_Byte6, TxMsg2_Byte7, TxMsg2_Byte8, TxMsg3_TransactionNumber, TxMsg3_CobId, TxMsg3_Byte1, TxMsg3_Byte2, TxMsg3_Byte3, TxMsg3_Byte4, TxMsg3_Byte5, TxMsg3_Byte6, TxMsg3_Byte7, TxMsg3_Byte8, TxMsg4_TransactionNumber, TxMsg4_CobId, TxMsg4_Byte1, TxMsg4_Byte2, TxMsg4_Byte3, TxMsg4_Byte4, TxMsg4_Byte5,
              TxMsg4_Byte6, TxMsg4_Byte7, TxMsg4_Byte8, TxMsg5_TransactionNumber, TxMsg5_CobId, TxMsg5_Byte1, TxMsg5_Byte2, TxMsg5_Byte3, TxMsg5_Byte4, TxMsg5_Byte5, TxMsg5_Byte6, TxMsg5_Byte7, TxMsg5_Byte8, TxMsg6_TransactionNumber, TxMsg6_CobId, TxMsg6_Byte1, TxMsg6_Byte2, TxMsg6_Byte3, TxMsg6_Byte4, TxMsg6_Byte5, TxMsg6_Byte6, TxMsg6_Byte7, TxMsg6_Byte8, TxMsg7_TransactionNumber, TxMsg7_CobId, TxMsg7_Byte1, TxMsg7_Byte2, TxMsg7_Byte3, TxMsg7_Byte4, TxMsg7_Byte5, TxMsg7_Byte6, TxMsg7_Byte7, TxMsg7_Byte8, TxMsg8_TransactionNumber, TxMsg8_CobId, TxMsg8_Byte1, TxMsg8_Byte2, TxMsg8_Byte3, TxMsg8_Byte4, TxMsg8_Byte5,
              TxMsg8_Byte6, TxMsg8_Byte7, TxMsg8_Byte8, CAN Control, TxCounter, RxCounter, NoOfRxMessages, TransactionNumber, RxMsg1_CobId, RxMsg1_Byte1, RxMsg1_Byte2, RxMsg1_Byte3, RxMsg1_Byte4, RxMsg1_Byte5, RxMsg1_Byte6, RxMsg1_Byte7, RxMsg1_Byte8, RxMsg2_CobId, RxMsg2_Byte1, RxMsg2_Byte2, RxMsg2_Byte3, RxMsg2_Byte4, RxMsg2_Byte5, RxMsg2_Byte6, RxMsg2_Byte7, RxMsg2_Byte8, RxMsg3_CobId, RxMsg3_Byte1, RxMsg3_Byte2, RxMsg3_Byte3, RxMsg3_Byte4, RxMsg3_Byte5, RxMsg3_Byte6, RxMsg3_Byte7, RxMsg3_Byte8, RxMsg4_CobId, RxMsg4_Byte1, RxMsg4_Byte2, RxMsg4_Byte3, RxMsg4_Byte4,
              RxMsg4_Byte5, RxMsg4_Byte6, RxMsg4_Byte7, RxMsg4_Byte8, RxMsg5_CobId, RxMsg5_Byte1, RxMsg5_Byte2, RxMsg5_Byte3, RxMsg5_Byte4, RxMsg5_Byte5, RxMsg5_Byte6, RxMsg5_Byte7, RxMsg5_Byte8, RxMsg6_CobId, RxMsg6_Byte1, RxMsg6_Byte2, RxMsg6_Byte3, RxMsg6_Byte4, RxMsg6_Byte5, RxMsg6_Byte6, RxMsg6_Byte7, RxMsg6_Byte8, RxMsg7_CobId, RxMsg7_Byte1, RxMsg7_Byte2, RxMsg7_Byte3, RxMsg7_Byte4, RxMsg7_Byte5, RxMsg7_Byte6, RxMsg7_Byte7, RxMsg7_Byte8, RxMsg8_CobId, RxMsg8_Byte1, RxMsg8_Byte2, RxMsg8_Byte3, RxMsg8_Byte4, RxMsg8_Byte5, RxMsg8_Byte6, RxMsg8_Byte7, RxMsg8_Byte8,
              CAN State, Align, RX Error Counter, TX Error Counter
          CANbus
              settings: NetID = 5
  libraries: VisuSymbols, 3.5.10.0 (System)
  text list GlobalTextList
*)

// Device/Application/can/canstruct/Can_BUS_8Inputs
TYPE Can_BUS_8Inputs :          //输入缓存结构 EL2721-8Message_IN
STRUCT
	TxCounter			: UINT;
	RxCounter			: UINT;
	NoOfRxMessages 	 	: UINT;
	TransactionNumber	: UINT;
	RXMsg				: ARRAY[1..8] OF Can_Bus_RXMsg_Buff;
	CAN_State			: UINT;
	Align				: UINT;
	RX_Error_Cnt		: BYTE;
	TX_Error_Cnt		: BYTE;
END_STRUCT
END_TYPE

// Device/Application/can/canstruct/Can_BUS_8Outputs
TYPE Can_BUS_8Outputs :		//输出缓存结构 EL2721-8Message_OUT
STRUCT
	TxCounter		: UINT;
	RxCounter		: UINT;
	NoOfTxMessages 	: UINT;
	TXMsg			: ARRAY[1..8] OF Can_Bus_TXMsg_Buff;
	CAN_Control		: UINT;
END_STRUCT
END_TYPE

// Device/Application/can/canstruct/Can_Bus_RXMsg_Buff
TYPE Can_Bus_RXMsg_Buff:
STRUCT
	RxMsg_CobId		: UINT;
	RxMsg_Byte  	: ARRAY[1..8] OF BYTE;
END_STRUCT
END_TYPE

// Device/Application/can/canstruct/Can_Bus_TXMsg_Buff
TYPE Can_Bus_TXMsg_Buff :
STRUCT
	TxMsg_TransactionNumber		: UINT;
	TxMsg_CobId					: UINT;
	TxMsg_Byte  				: ARRAY[1..8] OF BYTE;
END_STRUCT
END_TYPE

// Device/Application/can/canstruct/Can_baseframe
TYPE Can_baseframe :
STRUCT
	id		: UINT;
	data	: ARRAY[1..8] OF BYTE;
END_STRUCT
END_TYPE

// Device/Application/basestruct/CmdPercentSet
TYPE CmdPercentSet :
STRUCT
	extendPercent		:WORD;		//0-65535
	retractPercent		:WORD;		//0-65535
END_STRUCT
END_TYPE

// Device/Application/basestruct/SensorInfo
TYPE SensorInfo :
STRUCT
	
	position	:REAL;	//实时位移
	speed		:REAL;	//实时速度
	
	//记录最大最小位移值
	retractVal	:REAL;	//缩回到位值
	extendVal	:REAL;	//伸出到位值
	
END_STRUCT
END_TYPE

// Device/Application/basestruct/DeviceUnit
TYPE DeviceUnit :
STRUCT
		
	sensor			:SensorInfo;		//传感器参数
	ctrl			:DevPid;			//pid等计算控制执行参数	
	
	vector			:TargetDirect;		//指令运行方向 1-伸出 2-缩回 3-停止
	state			:DevStatus;			//设备状态 0-未知 1-运行 2-伸出到位 3-缩回到位 4-错误
	
	timeCounter		:INT;				//timeoutCounter超时计数器
	exeCounter		:INT;				//ExecuteCounter额外执行时间计数

	current			:ARRAY[1..2] OF WORD;	//电流mA	[i,j] -> 地轨挡板i的电流，j=1伸出电流，j=2缩回电流


END_STRUCT
END_TYPE

// Device/Application/basestruct/UIMode
TYPE UIMode :
STRUCT
	manualButtonSet			:BOOL;		//手动复位按钮模式
	usePID					:BOOL;		//使用pid
	autoEnable				:BOOL;		//自动使能
	manualPercentSet		:BOOL;		//手动设定比例量
	manualSetPid			:BOOL;		//手动调节pid参数，可通过pid测试界面设定目标位移值
	
	syncExt					:BOOL;		//同步伸
	syncRct					:BOOL;		//同步缩
	
	hydPowerOn				:BOOL;		//液压站开启 modbus 使用
	hydPowerOff				:BOOL;		//液压站关闭 modbus 使用
	hydPowerReset			:BOOL;		
END_STRUCT
END_TYPE

// Device/Application/basestruct/UIUnit
TYPE UIUnit :
STRUCT
	//cmd
	pwrEnable			:BOOL;		//比例阀使能   power-enable
	pwrPercent			:REAL;		//比例阀百分比 power-percent 0-100
	
	//button
	btnExtend			:BOOL;
	btnRetract			:BOOL;
	btnStop				:BOOL;
	btnLast				:TargetDirect;	//上次动作方向
	
	//info display
	name				:STRING;	//挡板名
	wname				:WSTRING;	//山河命名
	hzname				:WSTRING;	//hua zhong ming ming
	postion				:REAL;		//位移值
	speed				:REAL;
	extendPercent		:REAL;		//伸出百分比 extend-percent
	
	
	
END_STRUCT
END_TYPE

// Device/Application/basestruct/TargetDirect
{attribute 'qualified_only'}
{attribute 'strict'}
TYPE TargetDirect :
(
	extend 	:= 1,	//伸出
	
	retract := 2,	//缩回
	
	stop	:= 3	//停止
);
END_TYPE

// Device/Application/basestruct/DevStatus
{attribute 'qualified_only'}
{attribute 'strict'}
TYPE DevStatus :
(
	unknown 	:= 0,
	
	runing		:= 1,
	
	extended	:= 2,
	
	retracted	:= 3,
	
	error		:= 4
);
END_TYPE

// Device/Application/core/pid/PidParam
TYPE PidParam :
STRUCT
	Kp			:REAL;
	Ki			:REAL;
	Kd			:REAL;
	Set_Point	:REAL;
	Max_Val		:REAL;
	Max_ACC		:REAL;
	Act_Val		:REAL;
	Err			:REAL;
	OUT			:REAL;
END_STRUCT
END_TYPE

// Device/Application/core/pid/UiPid
TYPE UiPid :
STRUCT
	pos				:PidParam;			//位置pid参数
	spd				:PidParam;			//速度pid参数
	ff				:FeedForward;		//前馈参数

	level			:INT;				//1->地轨	2->天轨
	idx				:INT;				//挡板索引编号
	
	devSetPos		:REAL;				//设备中的设定位置点(用于观测)
	executeVal		:REAL;				//执行值(-100.0~+100.0)

	
	posBtn			:BOOL;			//位置控制按钮，按下实时更新交互参数
	rstPidBtn		:BOOL;			//reset pid param button重置pid参数按钮
	pwrPercent		:REAL;			//比例阀百分比 power-percent 0-100	
	
	
	
	
	extendBtn		:BOOL;
	retractBtn		:BOOL;
	stopBtn			:BOOL;


	
	
(*	posErr			:REAL;
	posOut			:REAL;
	spdErr			:REAL;
	spdOut			:REAL;*)	
END_STRUCT
END_TYPE

// Device/Application/core/pid/DevPid
TYPE DevPid :
STRUCT
	pos			:PidParam;			//位置pid参数
	spd			:PidParam;			//速度pid参数
	ff			:FeedForward;		//前馈参数
//	dp			:DynamicPlanning;	//规划参数
	exPct		:REAL;				//伸出默认比例量0-100
	rtPct		:REAL;				//缩回默认比例量0-100
	
	isError		:BOOL;				//当传感器数据为0时，报错并不执行pid
	
	extVal		:REAL;				//设定伸出位移值
	rtcVal		:REAL;				//设定缩回位移值
	
END_STRUCT
END_TYPE

// Device/Application/modbus/struct/mdbsStruct
TYPE mdbsStruct :
STRUCT
	request		:mdbsRequest;				//请求动作指令
	response	:mdbsResponse;			//响应动作指令-天地轨所有	
	
END_STRUCT
END_TYPE

// Device/Application/modbus/struct/mdbsRequest
TYPE mdbsRequest :	//所有请求动作指令数据
STRUCT
	startAddr		:WORD;					//解析起始地址->10
	length			:WORD;					//数据长度/字节->48
	data			:ARRAY[10..57] OF WORD;	//指令数据	
	
	arrNew		:ARRAY [1..4,0..15] OF BOOL;
	arrLast		:ARRAY [1..4,0..15] OF BOOL;

END_STRUCT
END_TYPE

// Device/Application/modbus/struct/mdbsResponse
TYPE mdbsResponse :	//所有响应状态数据回送
STRUCT
	startAddr		:WORD;							//解析起始地址->110
	length			:WORD;							//字节长度->210
	
	data			:ARRAY[110..319] OF WORD;		//位置数据

END_STRUCT
END_TYPE

// Device/Application/core/pid/FeedForward
TYPE FeedForward :
STRUCT
	
	pstThreshold	:REAL;	//正向设定阈值	
	pstKv			:REAL;
	pstKa			:REAL;
	pstKaa			:REAL;
	negThreshold	:REAL;	//反向设定阈值
	negKv			:REAL;
	negKa			:REAL;
	negKaa			:REAL;
	

	
//	pstFactor		:REAL;	//正向设定速度系数因子
//	negFactor		:REAL;	//反向设定速度系数因子


END_STRUCT
END_TYPE

// Device/Application/global/gController
{attribute 'qualified_only'}
VAR_GLOBAL
	//发送至SWMC的比例阀的控制指令
	sky		:ARRAY[0..10] OF CmdPercentSet;
	grd		:ARRAY[1..10] OF CmdPercentSet;
END_VAR

// Device/Application/global/gCan
{attribute 'qualified_only'}
VAR_GLOBAL
	C6TxMsg			AT%QW00		:Can_BUS_8Outputs;	
	C6RxMsg			AT%IW00		:Can_BUS_8Inputs;
	C6RxCounter			 	   	:UINT;
	
	C3TxMsg			AT%QW52		:Can_BUS_8Outputs;	
	C3RxMsg			AT%IW47		:Can_BUS_8Inputs;
	C3RxCounter			   	   	:UINT;

	C4TxMsg			AT%QW104	:Can_BUS_8Outputs;	
	C4RxMsg			AT%IW94		:Can_BUS_8Inputs;
	C4RxCounter				  	:UINT;

	C2TxMsg			AT%QW156	:Can_BUS_8Outputs;	
	C2RxMsg			AT%IW141	:Can_BUS_8Inputs;
	C2RxCounter			 	   	:UINT;
//(*	
	C1TxMsg			AT%QW208	:Can_BUS_8Outputs;	
	C1RxMsg			AT%IW188	:Can_BUS_8Inputs;
	C1RxCounter			   	   	:UINT;

	C5TxMsg			AT%QW260	:Can_BUS_8Outputs;	
	C5RxMsg			AT%IW235	:Can_BUS_8Inputs;
	C5RxCounter				  	:UINT;
//*)

END_VAR

// Device/Application/global/gDev
{attribute 'qualified_only'}
VAR_GLOBAL
	sky		:ARRAY[0..10] OF DeviceUnit;
	grd		:ARRAY[1..10] OF DeviceUnit;
END_VAR

// Device/Application/global/gUI
{attribute 'qualified_only'}
VAR_GLOBAL
	
	mode	:UIMode;					//模式设定

	sky		:ARRAY[0..10] OF UIUnit;	//挡板2组
	grd		:ARRAY[1..10] OF UIUnit;	//挡板1组
	
	pid		:UiPid;						//pid测试界面参数
	
	
	
END_VAR

// Device/Application/global/gModbus
{attribute 'qualified_only'}
VAR_GLOBAL CONSTANT
	g_modbusDataSizeMax	:  UINT:=65535; // 从机保持寄存器数量
END_VAR
VAR_GLOBAL
	srv				:mdbsStruct;		//modbus-service
	modbusBuffer	:ARRAY[0..g_modbusDataSizeMax] OF WORD;	//输入寄存器数据区	
END_VAR

// Device/Application/can/CanTx
PROGRAM CanTx
VAR
	count		:UINT;
END_VAR

count := count + 1;
IF count > 1000 THEN
	count := 1;
END_IF

C01_Tx();
C02_Tx();
C03_Tx();
C04_Tx();
C05_Tx();
C06_Tx();

METHOD C01_Tx
VAR_INPUT
END_VAR
VAR
	swmcIdSwtich		:UINT;
	sendData			:ARRAY[1..8] OF BYTE;
END_VAR

swmcIdSwtich := count MOD 2;
CASE swmcIdSwtich OF
	0:
		sendData[1] := WORD_TO_BYTE(gController.sky[3].extendPercent);
		sendData[2] := WORD_TO_BYTE(SHR(gController.sky[3].extendPercent,8));
		sendData[3] := WORD_TO_BYTE(gController.sky[3].retractPercent);
		sendData[4] := WORD_TO_BYTE(SHR(gController.sky[3].retractPercent,8));
		sendData[5] := WORD_TO_BYTE(gController.sky[4].extendPercent);
		sendData[6] := WORD_TO_BYTE(SHR(gController.sky[4].extendPercent,8));
		sendData[7] := WORD_TO_BYTE(gController.sky[4].retractPercent);
		sendData[8] := WORD_TO_BYTE(SHR(gController.sky[4].retractPercent,8));
		CAN_Send_Data_SWMC(1, 16#500,senddata);   //发送ID 0x460到C6
		
	1:
		sendData[1] := WORD_TO_BYTE(gController.sky[5].extendPercent);
		sendData[2] := WORD_TO_BYTE(SHR(gController.sky[5].extendPercent,8));
		sendData[3] := WORD_TO_BYTE(gController.sky[5].retractPercent);
		sendData[4] := WORD_TO_BYTE(SHR(gController.sky[5].retractPercent,8));
		sendData[5] := WORD_TO_BYTE(gController.sky[6].extendPercent);
		sendData[6] := WORD_TO_BYTE(SHR(gController.sky[6].extendPercent,8));
		sendData[7] := WORD_TO_BYTE(gController.sky[6].retractPercent);
		sendData[8] := WORD_TO_BYTE(SHR(gController.sky[6].retractPercent,8));
		CAN_Send_Data_SWMC(1, 16#501,senddata);   //发送ID 0x460到C6
		
		


END_CASE
END_METHOD

METHOD C02_Tx
VAR_INPUT
END_VAR
VAR
	swmcIdSwtich		:UINT;
	sendData			:ARRAY[1..8] OF BYTE;
END_VAR

swmcIdSwtich := count MOD 2;
CASE swmcIdSwtich OF
	0:
		sendData[1] := WORD_TO_BYTE(gController.sky[0].extendPercent);
		sendData[2] := WORD_TO_BYTE(SHR(gController.sky[0].extendPercent,8));
		sendData[3] := WORD_TO_BYTE(gController.sky[0].retractPercent);
		sendData[4] := WORD_TO_BYTE(SHR(gController.sky[0].retractPercent,8));
		sendData[5] := WORD_TO_BYTE(gController.sky[1].extendPercent);
		sendData[6] := WORD_TO_BYTE(SHR(gController.sky[1].extendPercent,8));
		sendData[7] := WORD_TO_BYTE(gController.sky[1].retractPercent);
		sendData[8] := WORD_TO_BYTE(SHR(gController.sky[1].retractPercent,8));
		CAN_Send_Data_SWMC(2, 16#510,senddata);   //发送ID 0x460到C6
		
	1:
		sendData[1] := WORD_TO_BYTE(gController.sky[2].extendPercent);
		sendData[2] := WORD_TO_BYTE(SHR(gController.sky[2].extendPercent,8));
		sendData[3] := WORD_TO_BYTE(gController.sky[2].retractPercent);
		sendData[4] := WORD_TO_BYTE(SHR(gController.sky[2].retractPercent,8));
		CAN_Send_Data_SWMC(2, 16#511,senddata);   //发送ID 0x460到C6
		
		


END_CASE
END_METHOD

METHOD C03_Tx
VAR_INPUT
END_VAR
VAR
	swmcIdSwtich		:UINT;
	sendData			:ARRAY[1..8] OF BYTE;
END_VAR

swmcIdSwtich := count MOD 2;
CASE swmcIdSwtich OF
	0:
		sendData[1] := WORD_TO_BYTE(gController.grd[3].extendPercent);
		sendData[2] := WORD_TO_BYTE(SHR(gController.grd[3].extendPercent,8));
		sendData[3] := WORD_TO_BYTE(gController.grd[3].retractPercent);
		sendData[4] := WORD_TO_BYTE(SHR(gController.grd[3].retractPercent,8));
		sendData[5] := WORD_TO_BYTE(gController.grd[4].extendPercent);
		sendData[6] := WORD_TO_BYTE(SHR(gController.grd[4].extendPercent,8));
		sendData[7] := WORD_TO_BYTE(gController.grd[4].retractPercent);
		sendData[8] := WORD_TO_BYTE(SHR(gController.grd[4].retractPercent,8));
		CAN_Send_Data_SWMC(3, 16#520,senddata);   //发送ID 0x460到C6
		
	1:
		sendData[1] := WORD_TO_BYTE(gController.grd[5].extendPercent);
		sendData[2] := WORD_TO_BYTE(SHR(gController.grd[5].extendPercent,8));
		sendData[3] := WORD_TO_BYTE(gController.grd[5].retractPercent);
		sendData[4] := WORD_TO_BYTE(SHR(gController.grd[5].retractPercent,8));
		sendData[5] := WORD_TO_BYTE(gController.grd[6].extendPercent);
		sendData[6] := WORD_TO_BYTE(SHR(gController.grd[6].extendPercent,8));
		sendData[7] := WORD_TO_BYTE(gController.grd[6].retractPercent);
		sendData[8] := WORD_TO_BYTE(SHR(gController.grd[6].retractPercent,8));
		CAN_Send_Data_SWMC(3, 16#521,senddata);   //发送ID 0x460到C6
		
		


END_CASE
END_METHOD

METHOD C04_Tx
VAR_INPUT
END_VAR
VAR
	swmcIdSwtich		:UINT;
	sendData			:ARRAY[1..8] OF BYTE;
END_VAR

swmcIdSwtich := count MOD 2;
CASE swmcIdSwtich OF
	0:
		sendData[1] := WORD_TO_BYTE(gController.grd[1].extendPercent);
		sendData[2] := WORD_TO_BYTE(SHR(gController.grd[1].extendPercent,8));
		sendData[3] := WORD_TO_BYTE(gController.grd[1].retractPercent);
		sendData[4] := WORD_TO_BYTE(SHR(gController.grd[1].retractPercent,8));
		sendData[5] := WORD_TO_BYTE(gController.grd[2].extendPercent);
		sendData[6] := WORD_TO_BYTE(SHR(gController.grd[2].extendPercent,8));
		sendData[7] := WORD_TO_BYTE(gController.grd[2].retractPercent);
		sendData[8] := WORD_TO_BYTE(SHR(gController.grd[2].retractPercent,8));
		CAN_Send_Data_SWMC(4, 16#530,senddata);   //发送ID 0x460到C6
		
		
		


END_CASE
END_METHOD

METHOD C05_Tx
VAR_INPUT
END_VAR
VAR
	swmcIdSwtich		:UINT;
	sendData			:ARRAY[1..8] OF BYTE;
END_VAR

swmcIdSwtich := count MOD 2;
CASE swmcIdSwtich OF
	0:
		sendData[1] := WORD_TO_BYTE(gController.sky[7].extendPercent);
		sendData[2] := WORD_TO_BYTE(SHR(gController.sky[7].extendPercent,8));
		sendData[3] := WORD_TO_BYTE(gController.sky[7].retractPercent);
		sendData[4] := WORD_TO_BYTE(SHR(gController.sky[7].retractPercent,8));
		sendData[5] := WORD_TO_BYTE(gController.sky[8].extendPercent);
		sendData[6] := WORD_TO_BYTE(SHR(gController.sky[8].extendPercent,8));
		sendData[7] := WORD_TO_BYTE(gController.sky[8].retractPercent);
		sendData[8] := WORD_TO_BYTE(SHR(gController.sky[8].retractPercent,8));
		CAN_Send_Data_SWMC(5, 16#540,senddata);   //发送ID 0x460到C6	
	1:
		sendData[1] := WORD_TO_BYTE(gController.sky[9].extendPercent);
		sendData[2] := WORD_TO_BYTE(SHR(gController.sky[9].extendPercent,8));
		sendData[3] := WORD_TO_BYTE(gController.sky[9].retractPercent);
		sendData[4] := WORD_TO_BYTE(SHR(gController.sky[9].retractPercent,8));
		sendData[5] := WORD_TO_BYTE(gController.sky[10].extendPercent);
		sendData[6] := WORD_TO_BYTE(SHR(gController.sky[10].extendPercent,8));
		sendData[7] := WORD_TO_BYTE(gController.sky[10].retractPercent);
		sendData[8] := WORD_TO_BYTE(SHR(gController.sky[10].retractPercent,8));
		CAN_Send_Data_SWMC(5, 16#541,senddata);   //发送ID 0x460到C6		

END_CASE
END_METHOD

METHOD C06_Tx
VAR_INPUT
END_VAR
VAR
	swmcIdSwtich		:UINT;
	sendData			:ARRAY[1..8] OF BYTE;
END_VAR

swmcIdSwtich := count MOD 2;
CASE swmcIdSwtich OF
	0:
		sendData[1] := WORD_TO_BYTE(gController.grd[7].extendPercent);
		sendData[2] := WORD_TO_BYTE(SHR(gController.grd[7].extendPercent,8));
		sendData[3] := WORD_TO_BYTE(gController.grd[7].retractPercent);
		sendData[4] := WORD_TO_BYTE(SHR(gController.grd[7].retractPercent,8));
		sendData[5] := WORD_TO_BYTE(gController.grd[8].extendPercent);
		sendData[6] := WORD_TO_BYTE(SHR(gController.grd[8].extendPercent,8));
		sendData[7] := WORD_TO_BYTE(gController.grd[8].retractPercent);
		sendData[8] := WORD_TO_BYTE(SHR(gController.grd[8].retractPercent,8));
		CAN_Send_Data_SWMC(6, 16#550,senddata);   //发送ID 0x460到C6
		
	1:
		sendData[1] := WORD_TO_BYTE(gController.grd[9].extendPercent);
		sendData[2] := WORD_TO_BYTE(SHR(gController.grd[9].extendPercent,8));
		sendData[3] := WORD_TO_BYTE(gController.grd[9].retractPercent);
		sendData[4] := WORD_TO_BYTE(SHR(gController.grd[9].retractPercent,8));
		sendData[5] := WORD_TO_BYTE(gController.grd[10].extendPercent);
		sendData[6] := WORD_TO_BYTE(SHR(gController.grd[10].extendPercent,8));
		sendData[7] := WORD_TO_BYTE(gController.grd[10].retractPercent);
		sendData[8] := WORD_TO_BYTE(SHR(gController.grd[10].retractPercent,8));
		CAN_Send_Data_SWMC(6, 16#551,senddata);   //发送ID 0x460到C6
		
END_CASE
END_METHOD

END_PROGRAM

// Device/Application/can/CAN_Send_Data_SWMC
FUNCTION CAN_Send_Data_SWMC : BOOL
VAR_INPUT
	SWMC_ID : UINT;
	id 		: UINT;
	data	: ARRAY[1..8] OF BYTE;
END_VAR
VAR
	
END_VAR

CASE  SWMC_ID OF

	1:
		gCan.C1TxMsg.TXMsg[1].TxMsg_CobId 	:= 8 + 32 * id;
	  	gCan.C1TxMsg.TXMsg[1].TxMsg_Byte 	:= data;
	   	gCan.C1TxMsg.NoOfTxMessages			:= 1;
	   	gCan.C1TxMsg.TxCounter 				:= gCan.C1TxMsg.TxCounter +1;	
	2:
		gCan.C2TxMsg.TXMsg[1].TxMsg_CobId 	:= 8 + 32 * id;
	  	gCan.C2TxMsg.TXMsg[1].TxMsg_Byte 	:= data;
	   	gCan.C2TxMsg.NoOfTxMessages			:= 1;
	   	gCan.C2TxMsg.TxCounter 				:= gCan.C2TxMsg.TxCounter +1;	
	3:
		gCan.C3TxMsg.TXMsg[1].TxMsg_CobId 	:= 8 + 32 * id;
	  	gCan.C3TxMsg.TXMsg[1].TxMsg_Byte 	:= data;
	   	gCan.C3TxMsg.NoOfTxMessages			:= 1;
	   	gCan.C3TxMsg.TxCounter 				:= gCan.C3TxMsg.TxCounter +1;
	4:
		gCan.C4TxMsg.TXMsg[1].TxMsg_CobId 	:= 8 + 32 * id;
	  	gCan.C4TxMsg.TXMsg[1].TxMsg_Byte 	:= data;
	   	gCan.C4TxMsg.NoOfTxMessages			:= 1;
	   	gCan.C4TxMsg.TxCounter 				:= gCan.C4TxMsg.TxCounter +1;
	//(*
	5:
		gCan.C5TxMsg.TXMsg[1].TxMsg_CobId 	:= 8 + 32 * id;
	  	gCan.C5TxMsg.TXMsg[1].TxMsg_Byte 	:= data;
	   	gCan.C5TxMsg.NoOfTxMessages			:= 1;
	   	gCan.C5TxMsg.TxCounter 				:= gCan.C5TxMsg.TxCounter +1;
	6:
		gCan.C6TxMsg.TXMsg[1].TxMsg_CobId 	:= 8 + 32 * id;
	  	gCan.C6TxMsg.TXMsg[1].TxMsg_Byte 	:= data;
	   	gCan.C6TxMsg.NoOfTxMessages			:= 1;
	   	gCan.C6TxMsg.TxCounter 				:= gCan.C6TxMsg.TxCounter +1;
	//*)

END_CASE

END_FUNCTION

// Device/Application/can/CanRx
PROGRAM CanRx
VAR
	count		:UINT;
END_VAR

count := count + 1;
IF count > 1000 THEN
	count := 1;
END_IF

C01_Rx();
C02_Rx();
C03_Rx();
C04_Rx();
C05_Rx();
C06_Rx();

METHOD C01_Rx
VAR_INPUT
END_VAR
VAR
	frame	 	    :Can_baseframe;
	I				:UINT;
	fId				:UINT;
	pos				:WORD;
	spd				:WORD;
END_VAR
IF gCan.C1RxMsg.RxCounter <>  gCan.C1RxCounter THEN    //接收到新的数据
	FOR I := 1 TO gCan.C1RxMsg.NoOfRxMessages DO
		frame := CAN_Read_Data_SWMC(1,I);
		fId := frame.id;
		CASE fId OF
			16#600:
				pos := BYTE_TO_WORD(frame.data[ 1 ]) OR SHL(BYTE_TO_WORD(frame.data[ 2 ]),8);
				gDev.sky[4].sensor.position := pos * 0.1;
				pos := BYTE_TO_WORD(frame.data[ 3 ]) OR SHL(BYTE_TO_WORD(frame.data[ 4 ]),8);
				gDev.sky[5].sensor.position := pos * 0.1;
				pos := BYTE_TO_WORD(frame.data[ 5 ]) OR SHL(BYTE_TO_WORD(frame.data[ 6 ]),8);
				gDev.sky[6].sensor.position := pos * 0.1;
				pos := BYTE_TO_WORD(frame.data[ 7 ]) OR SHL(BYTE_TO_WORD(frame.data[ 8 ]),8);
				gDev.sky[3].sensor.position := pos * 0.1;
			16#601:
				spd := BYTE_TO_WORD(frame.data[ 1 ]) OR SHL(BYTE_TO_WORD(frame.data[ 2 ]),8);
				gDev.sky[4].sensor.speed := INT_TO_REAL(WORD_TO_INT(spd));
				spd := BYTE_TO_WORD(frame.data[ 3 ]) OR SHL(BYTE_TO_WORD(frame.data[ 4 ]),8);
				gDev.sky[5].sensor.speed := INT_TO_REAL(WORD_TO_INT(spd));
				spd := BYTE_TO_WORD(frame.data[ 5 ]) OR SHL(BYTE_TO_WORD(frame.data[ 6 ]),8);
				gDev.sky[6].sensor.speed := INT_TO_REAL(WORD_TO_INT(spd));
				spd := BYTE_TO_WORD(frame.data[ 7 ]) OR SHL(BYTE_TO_WORD(frame.data[ 8 ]),8);
				gDev.sky[3].sensor.speed := INT_TO_REAL(WORD_TO_INT(spd));
		END_CASE

	END_FOR
	gCan.C1RxCounter := gCan.C1RxMsg.RxCounter;
END_IF
END_METHOD

METHOD C02_Rx
VAR_INPUT
END_VAR
VAR
	frame	 	    :Can_baseframe;
	I				:UINT;
	fId				:UINT;
	pos				:WORD;
	spd				:WORD;
END_VAR
IF gCan.C2RxMsg.RxCounter <>  gCan.C2RxCounter THEN    //接收到新的数据
	FOR I := 1 TO gCan.C2RxMsg.NoOfRxMessages DO
		frame := CAN_Read_Data_SWMC(2,I);
		fId := frame.id;
		CASE fId OF
			16#610:
				pos := BYTE_TO_WORD(frame.data[ 1 ]) OR SHL(BYTE_TO_WORD(frame.data[ 2 ]),8);
				gDev.sky[0].sensor.position := pos * 0.1;
				pos := BYTE_TO_WORD(frame.data[ 3 ]) OR SHL(BYTE_TO_WORD(frame.data[ 4 ]),8);
				gDev.sky[1].sensor.position := pos * 0.1;
				pos := BYTE_TO_WORD(frame.data[ 5 ]) OR SHL(BYTE_TO_WORD(frame.data[ 6 ]),8);
				gDev.sky[2].sensor.position := pos * 0.1;
	
			16#611:
				spd := BYTE_TO_WORD(frame.data[ 1 ]) OR SHL(BYTE_TO_WORD(frame.data[ 2 ]),8);
				gDev.sky[0].sensor.speed := INT_TO_REAL(WORD_TO_INT(spd));
				spd := BYTE_TO_WORD(frame.data[ 3 ]) OR SHL(BYTE_TO_WORD(frame.data[ 4 ]),8);
				gDev.sky[1].sensor.speed := INT_TO_REAL(WORD_TO_INT(spd));
				spd := BYTE_TO_WORD(frame.data[ 5 ]) OR SHL(BYTE_TO_WORD(frame.data[ 6 ]),8);
				gDev.sky[2].sensor.speed := INT_TO_REAL(WORD_TO_INT(spd));
		END_CASE
	END_FOR
	gCan.C2RxCounter := gCan.C2RxMsg.RxCounter;
END_IF
END_METHOD

METHOD C03_Rx
VAR_INPUT
END_VAR
VAR
	frame	 	    :Can_baseframe;
	I				:UINT;
	fId				:UINT;
	pos				:WORD;
	spd				:WORD;
	cur				:WORD;	//current
END_VAR
IF gCan.C3RxMsg.RxCounter <>  gCan.C3RxCounter THEN    //接收到新的数据
	FOR I := 1 TO gCan.C3RxMsg.NoOfRxMessages DO
		frame := CAN_Read_Data_SWMC(3,I);
		fId := frame.id;
		CASE fId OF
			16#620:
				pos := BYTE_TO_WORD(frame.data[ 1 ]) OR SHL(BYTE_TO_WORD(frame.data[ 2 ]),8);
				gDev.grd[5].sensor.position := pos * 0.1;
				pos := BYTE_TO_WORD(frame.data[ 3 ]) OR SHL(BYTE_TO_WORD(frame.data[ 4 ]),8);
				gDev.grd[6].sensor.position := pos * 0.1;
				pos := BYTE_TO_WORD(frame.data[ 5 ]) OR SHL(BYTE_TO_WORD(frame.data[ 6 ]),8);
				gDev.grd[3].sensor.position := pos * 0.1;
				pos := BYTE_TO_WORD(frame.data[ 7 ]) OR SHL(BYTE_TO_WORD(frame.data[ 8 ]),8);
				gDev.grd[4].sensor.position := pos * 0.1;
			16#621:
				spd := BYTE_TO_WORD(frame.data[ 1 ]) OR SHL(BYTE_TO_WORD(frame.data[ 2 ]),8);
				gDev.grd[5].sensor.speed := INT_TO_REAL(WORD_TO_INT(spd));
				spd := BYTE_TO_WORD(frame.data[ 3 ]) OR SHL(BYTE_TO_WORD(frame.data[ 4 ]),8);
				gDev.grd[6].sensor.speed := INT_TO_REAL(WORD_TO_INT(spd));
				spd := BYTE_TO_WORD(frame.data[ 5 ]) OR SHL(BYTE_TO_WORD(frame.data[ 6 ]),8);
				gDev.grd[3].sensor.speed := INT_TO_REAL(WORD_TO_INT(spd));
				spd := BYTE_TO_WORD(frame.data[ 7 ]) OR SHL(BYTE_TO_WORD(frame.data[ 8 ]),8);
				gDev.grd[4].sensor.speed := INT_TO_REAL(WORD_TO_INT(spd));	
			16#622:
				cur := BYTE_TO_WORD(frame.data[ 1 ]) OR SHL(BYTE_TO_WORD(frame.data[ 2 ]),8);
				gDev.grd[3].current[1] := cur;
				cur := BYTE_TO_WORD(frame.data[ 3 ]) OR SHL(BYTE_TO_WORD(frame.data[ 4 ]),8);
				gDev.grd[3].current[2] := cur;
				cur := BYTE_TO_WORD(frame.data[ 5 ]) OR SHL(BYTE_TO_WORD(frame.data[ 6 ]),8);
				gDev.grd[4].current[1] := cur;
				cur := BYTE_TO_WORD(frame.data[ 7 ]) OR SHL(BYTE_TO_WORD(frame.data[ 8 ]),8);
				gDev.grd[4].current[2] := cur;
			16#623:
				cur := BYTE_TO_WORD(frame.data[ 1 ]) OR SHL(BYTE_TO_WORD(frame.data[ 2 ]),8);
				gDev.grd[5].current[1] := cur;
				cur := BYTE_TO_WORD(frame.data[ 3 ]) OR SHL(BYTE_TO_WORD(frame.data[ 4 ]),8);
				gDev.grd[5].current[2] := cur;
				cur := BYTE_TO_WORD(frame.data[ 5 ]) OR SHL(BYTE_TO_WORD(frame.data[ 6 ]),8);
				gDev.grd[6].current[1] := cur;
				cur := BYTE_TO_WORD(frame.data[ 7 ]) OR SHL(BYTE_TO_WORD(frame.data[ 8 ]),8);
				gDev.grd[6].current[2] := cur;
				
				
				
		END_CASE
	END_FOR
	gCan.C3RxCounter := gCan.C3RxMsg.RxCounter;
END_IF
END_METHOD

METHOD C04_Rx
VAR_INPUT
END_VAR
VAR
	frame	 	    :Can_baseframe;
	I				:UINT;
	fId				:UINT;
	pos				:WORD;
	spd				:WORD;
	
END_VAR
IF gCan.C4RxMsg.RxCounter <>  gCan.C4RxCounter THEN    //接收到新的数据
	FOR I := 1 TO gCan.C4RxMsg.NoOfRxMessages DO
		frame := CAN_Read_Data_SWMC(4,I);
		fId := frame.id;
		CASE fId OF
			16#630:
				pos := BYTE_TO_WORD(frame.data[ 1 ]) OR SHL(BYTE_TO_WORD(frame.data[ 2 ]),8);
				gDev.grd[1].sensor.position := pos * 0.1;
				pos := BYTE_TO_WORD(frame.data[ 3 ]) OR SHL(BYTE_TO_WORD(frame.data[ 4 ]),8);
				gDev.grd[2].sensor.position := pos * 0.1;
	
			16#631:
				spd := BYTE_TO_WORD(frame.data[ 1 ]) OR SHL(BYTE_TO_WORD(frame.data[ 2 ]),8);
				gDev.grd[1].sensor.speed := INT_TO_REAL(WORD_TO_INT(spd));
				spd := BYTE_TO_WORD(frame.data[ 3 ]) OR SHL(BYTE_TO_WORD(frame.data[ 4 ]),8);
				gDev.grd[2].sensor.speed := INT_TO_REAL(WORD_TO_INT(spd));
		END_CASE
	END_FOR
	gCan.C4RxCounter := gCan.C4RxMsg.RxCounter;
END_IF
END_METHOD

METHOD C05_Rx
VAR_INPUT
END_VAR
VAR
	frame	 	    :Can_baseframe;
	I				:UINT;
	fId				:UINT;
	pos				:WORD;	//位置
	spd				:WORD;	//速度
END_VAR
IF gCan.C5RxMsg.RxCounter <>  gCan.C5RxCounter THEN    //接收到新的数据
	FOR I := 1 TO gCan.C5RxMsg.NoOfRxMessages DO
		frame := CAN_Read_Data_SWMC(5,I);
		fId := frame.id;
		CASE fId OF
			16#640:
				pos := BYTE_TO_WORD(frame.data[ 1 ]) OR SHL(BYTE_TO_WORD(frame.data[ 2 ]),8);
				gDev.sky[7].sensor.position := pos * 0.1;
				pos := BYTE_TO_WORD(frame.data[ 3 ]) OR SHL(BYTE_TO_WORD(frame.data[ 4 ]),8);
				gDev.sky[8].sensor.position := pos * 0.1;
				pos := BYTE_TO_WORD(frame.data[ 5 ]) OR SHL(BYTE_TO_WORD(frame.data[ 6 ]),8);
				gDev.sky[9].sensor.position := pos * 0.1;
				pos := BYTE_TO_WORD(frame.data[ 7 ]) OR SHL(BYTE_TO_WORD(frame.data[ 8 ]),8);
				gDev.sky[10].sensor.position := pos * 0.1;
			16#641:
				spd := BYTE_TO_WORD(frame.data[ 1 ]) OR SHL(BYTE_TO_WORD(frame.data[ 2 ]),8);
				gDev.sky[7].sensor.speed := INT_TO_REAL(WORD_TO_INT(spd));
				spd := BYTE_TO_WORD(frame.data[ 3 ]) OR SHL(BYTE_TO_WORD(frame.data[ 4 ]),8);
				gDev.sky[8].sensor.speed := INT_TO_REAL(WORD_TO_INT(spd));
				spd := BYTE_TO_WORD(frame.data[ 5 ]) OR SHL(BYTE_TO_WORD(frame.data[ 6 ]),8);
				gDev.sky[9].sensor.speed := INT_TO_REAL(WORD_TO_INT(spd));
				spd := BYTE_TO_WORD(frame.data[ 7 ]) OR SHL(BYTE_TO_WORD(frame.data[ 8 ]),8);
				gDev.sky[10].sensor.speed := INT_TO_REAL(WORD_TO_INT(spd));	
		END_CASE

	END_FOR
	gCan.C5RxCounter := gCan.C5RxMsg.RxCounter;
END_IF
END_METHOD

METHOD C06_Rx
VAR_INPUT
END_VAR
VAR
	frame	 	    :Can_baseframe;
	I				:UINT;
	fId				:UINT;
	pos				:WORD;	//位置
	spd				:WORD;	//速度
END_VAR
IF gCan.C6RxMsg.RxCounter <>  gCan.C6RxCounter THEN    //接收到新的数据
	FOR I := 1 TO gCan.C6RxMsg.NoOfRxMessages DO
		frame := CAN_Read_Data_SWMC(6,I);
		fId := frame.id;
		CASE fId OF
			16#650:
				pos := BYTE_TO_WORD(frame.data[ 1 ]) OR SHL(BYTE_TO_WORD(frame.data[ 2 ]),8);
				gDev.grd[7].sensor.position := pos * 0.1;
				pos := BYTE_TO_WORD(frame.data[ 3 ]) OR SHL(BYTE_TO_WORD(frame.data[ 4 ]),8);
				gDev.grd[8].sensor.position := pos * 0.1;
				pos := BYTE_TO_WORD(frame.data[ 5 ]) OR SHL(BYTE_TO_WORD(frame.data[ 6 ]),8);
				gDev.grd[9].sensor.position := pos * 0.1;
				pos := BYTE_TO_WORD(frame.data[ 7 ]) OR SHL(BYTE_TO_WORD(frame.data[ 8 ]),8);
				gDev.grd[10].sensor.position := pos * 0.1;
			16#651:
				spd := BYTE_TO_WORD(frame.data[ 1 ]) OR SHL(BYTE_TO_WORD(frame.data[ 2 ]),8);
				gDev.grd[7].sensor.speed := INT_TO_REAL(WORD_TO_INT(spd));
				spd := BYTE_TO_WORD(frame.data[ 3 ]) OR SHL(BYTE_TO_WORD(frame.data[ 4 ]),8);
				gDev.grd[8].sensor.speed := INT_TO_REAL(WORD_TO_INT(spd));
				spd := BYTE_TO_WORD(frame.data[ 5 ]) OR SHL(BYTE_TO_WORD(frame.data[ 6 ]),8);
				gDev.grd[9].sensor.speed := INT_TO_REAL(WORD_TO_INT(spd));
				spd := BYTE_TO_WORD(frame.data[ 7 ]) OR SHL(BYTE_TO_WORD(frame.data[ 8 ]),8);
				gDev.grd[10].sensor.speed := INT_TO_REAL(WORD_TO_INT(spd));	
		END_CASE
	END_FOR
	gCan.C6RxCounter := gCan.C6RxMsg.RxCounter;
END_IF
END_METHOD

END_PROGRAM

// Device/Application/can/CAN_Read_Data_SWMC
FUNCTION CAN_Read_Data_SWMC : Can_baseframe
VAR_INPUT
	SWMC_ID	 :UINT;		//接收SWMC控制ID
	I	 	 :UINT;      //接收缓冲区域
END_VAR
VAR
	frame :Can_baseframe;
END_VAR

CASE  SWMC_ID OF

	1:                       //SWMC-C1
		frame.id 	:= (gCan.C1RxMsg.RXMsg[I].RxMsg_CobId-8)/32;
		frame.data 	:= gCan.C1RxMsg.RXMsg[I].RxMsg_Byte;				
	2:                       //SWMC-C2
		frame.id 	:= (gCan.C2RxMsg.RXMsg[I].RxMsg_CobId-8)/32;
		frame.data 	:= gCan.C2RxMsg.RXMsg[I].RxMsg_Byte;
	3:						//SWMC-C3
		frame.id 	:= (gCan.C3RxMsg.RXMsg[I].RxMsg_CobId-8)/32;
		frame.data 	:= gCan.C3RxMsg.RXMsg[I].RxMsg_Byte;	
	4:                       //SWMC-C4
		frame.id 	:= (gCan.C4RxMsg.RXMsg[I].RxMsg_CobId-8)/32;
		frame.data 	:= gCan.C4RxMsg.RXMsg[I].RxMsg_Byte;				
	//(*
	5:                       //SWMC-C5
		frame.id 	:= (gCan.C5RxMsg.RXMsg[I].RxMsg_CobId-8)/32;
		frame.data 	:= gCan.C5RxMsg.RXMsg[I].RxMsg_Byte;
	6:						//SWMC-C6
		frame.id 	:= (gCan.C6RxMsg.RXMsg[I].RxMsg_CobId-8)/32;
		frame.data 	:= gCan.C6RxMsg.RXMsg[I].RxMsg_Byte;	
		//*)
	ELSE				//Other
		frame.id := 0;
		frame.data[1] := 0;
		frame.data[2] := 0;
		frame.data[3] := 0;
		frame.data[4] := 0;
		frame.data[5] := 0;
		frame.data[6] := 0;
		frame.data[7] := 0;
		frame.data[8] := 0;
END_CASE
Can_Read_data_SWMC := frame;

END_FUNCTION

// Device/Application/core/Barrier
PROGRAM Barrier
VAR
	bInit			:BOOL:=TRUE;
	initCount		:INT:= 100 * 2;		//2s后开始初始化，执行
	timeout			:INT:= 100 * 16;	//10ms间隔时 is 15 second
	timeexe			:INT:= 100 * 8;		//需要停止时，额外执行指令时间
	cmdExecutor0	:CommandExecutor0;
	cmdExecutor		:CommandExecutor;
	grdPid			:ARRAY[1..10] OF grdPosCtrl;
	skyPid			:ARRAY[0..10] OF skyPosCtrl;
	resetPidParam	:BOOL;							//pid参数复位
	pidMode			:BOOL;							//使用pid控制
	autoButtonMode	:BOOL;							//手动复位按钮
	autoEnableMode	:BOOL;							//有动作时使能自动开启
	autoPctMode		:BOOL;
	manualPidPrmSet	:BOOL;							//manualPidParamSet,手动设定pid位置参数

	gi				:INT;			//ground-i
	si				:INT;			//sky-i

	level			:INT;			//1->地轨	2->天轨
	idx				:INT := -1 ;	//挡板索引编号
END_VAR

//初始化
IF initCount = 0 THEN
	IF bInit THEN
		initialize();
		initializePid();
		bInit := FALSE;
	END_IF
ELSE
	initCount := initCount - 1;
	RETURN;	
END_IF

//指令执行
pidTestUi();

IF pidMode THEN
	pidCalc();
	pidExecute();
ELSE
	IF autoPctMode THEN setExecutePercent(); END_IF
	manualExecute();
END_IF	

//界面交互  
interfaceAct();

//状态更新
updateStatus(error := 1);

//复位按钮模式/
IF autoButtonMode THEN
	autoResetButton();
END_IF
IF autoEnableMode THEN
	autoEnable();
END_IF

METHOD updateStatus
VAR_INPUT
		error			:REAL;
END_VAR

VAR 
		devstat			:DevStatus;	
		needStop		:BOOL;	
END_VAR
FOR gi := 1 TO 10 DO
	//计数器
	IF gDev.grd[gi].state = DevStatus.runing THEN
		gDev.grd[gi].timeCounter := gDev.grd[gi].timeCounter + 1;	
		IF gDev.grd[gi].timeCounter > timeout THEN		//超时更改状态
			gDev.grd[gi].timeCounter := 0;
			gDev.grd[gi].state := DevStatus.error;
			gDev.grd[gi].vector := TargetDirect.stop;
		END_IF
	END_IF
	IF gDev.grd[gi].vector = TargetDirect.stop THEN
		gDev.grd[gi].timeCounter := 0;
	END_IF
	devstat := updateDevStatus(1, gi, error);//若伸/缩到位更新状态，否则不更新
	//伸缩到位时接收到伸缩指令执行exeCounter对应的时间
	(*
	needStop := (gDev.grd[gi].state = DevStatus.extended AND gDev.grd[gi].vector = TargetDirect.extend) OR 
			 	(gDev.grd[gi].state = DevStatus.retracted AND gDev.grd[gi].vector = TargetDirect.retract) ;	
	IF needStop THEN
		gDev.grd[gi].exeCounter := gDev.grd[gi].exeCounter + 1;
		IF gDev.grd[gi].exeCounter > timeexe THEN
			gDev.grd[gi].exeCounter := 0;
			gDev.grd[gi].timeCounter := 0;
			gDev.grd[gi].state := DevStatus.error;
			gDev.grd[gi].vector := TargetDirect.stop;
		END_IF
	ELSE
		gDev.grd[gi].exeCounter := 0;
	END_IF
	*)
END_FOR


FOR si := 0 TO 10 DO
	//计数器
	IF gDev.sky[si].state = DevStatus.runing THEN
		gDev.sky[si].timeCounter := gDev.sky[si].timeCounter + 1;	
		IF gDev.sky[si].timeCounter > timeout THEN		//超时更改状态
			gDev.sky[si].timeCounter := 0;
			gDev.sky[si].state := DevStatus.error;
			gDev.sky[si].vector := TargetDirect.stop;
		END_IF
	END_IF
	IF gDev.sky[si].vector = TargetDirect.stop THEN
		gDev.sky[si].timeCounter := 0;
	END_IF
	devstat := updateDevStatus(2, si, error);	//若伸/缩到位更新状态，否则不更新
	(*
	//伸缩到位时接收到伸缩指令执行exeCounter对应的时间
	needStop := (gDev.sky[si].state = DevStatus.extended AND gDev.sky[si].vector = TargetDirect.extend)
			 OR (gDev.sky[si].state = DevStatus.retracted AND gDev.sky[si].vector = TargetDirect.retract);
	IF needStop THEN
		gDev.sky[si].exeCounter := gDev.sky[si].exeCounter + 1;
		IF gDev.sky[si].exeCounter > timeexe THEN
			gDev.sky[si].exeCounter := 0;
			gDev.sky[si].timeCounter := 0;
			gDev.sky[si].state := DevStatus.error;
			gDev.sky[si].vector := TargetDirect.stop;
		END_IF
	ELSE
		gDev.sky[si].exeCounter := 0;
	END_IF
	*)
END_FOR
END_METHOD

ACTION initialize:
//默认自动使能
gUI.mode.autoEnable	:= TRUE;
gUI.mode.usePID := TRUE;

//initialize boundary val
	//ground
	gDev.grd[	1	].sensor.retractVal	:=	4.4	;		gDev.grd[	1	].sensor.extendVal	:=	108 	;
	gDev.grd[	2	].sensor.retractVal	:=	3.5	;		gDev.grd[	2	].sensor.extendVal	:=	113.4	;
	gDev.grd[	3	].sensor.retractVal	:=	4.1	;		gDev.grd[	3	].sensor.extendVal	:=	110 	;
	gDev.grd[	4	].sensor.retractVal	:=	1	;		gDev.grd[	4	].sensor.extendVal	:=	112.3	;		//结构问题暂不动
	gDev.grd[	5	].sensor.retractVal	:=	4.0	;		gDev.grd[	5	].sensor.extendVal	:=	107.1-0.5	;
	gDev.grd[	6	].sensor.retractVal	:=	3.5	;		gDev.grd[	6	].sensor.extendVal	:=	110.5	;
	gDev.grd[	7	].sensor.retractVal	:=	5	;		gDev.grd[	7	].sensor.extendVal	:=	109.7   ;
	gDev.grd[	8	].sensor.retractVal	:=	4.8	;		gDev.grd[	8	].sensor.extendVal	:=	109.2	;
	gDev.grd[	9	].sensor.retractVal	:=	3.2	;		gDev.grd[	9	].sensor.extendVal	:=	108 -0.5 	;
	gDev.grd[	10	].sensor.retractVal	:=	6.9	;		gDev.grd[	10	].sensor.extendVal	:=	112 	;
(*	
	gDev.grd[	7	].sensor.retractVal	:=	3.6	;		gDev.grd[	7	].sensor.extendVal	:=	108.3	;
	gDev.grd[	8	].sensor.retractVal	:=	3.5	;		gDev.grd[	8	].sensor.extendVal	:=	113.1	;
	gDev.grd[	9	].sensor.retractVal	:=	3.2	;		gDev.grd[	9	].sensor.extendVal	:=	107.3	;
	gDev.grd[	10	].sensor.retractVal	:=	3.4	;		gDev.grd[	10	].sensor.extendVal	:=	113.5	;*)

	//sky	
	gDev.sky[	0	].sensor.retractVal	:=	3.7	;		gDev.sky[	0	].sensor.extendVal	:=	213.6	;
	gDev.sky[	1	].sensor.retractVal	:=	8.8	;		gDev.sky[	1	].sensor.extendVal	:=	113.1	;
	gDev.sky[	2	].sensor.retractVal	:=	3.5	;		gDev.sky[	2	].sensor.extendVal	:=	113.0	;
	gDev.sky[	3	].sensor.retractVal	:=	3.5	;		gDev.sky[	3	].sensor.extendVal	:=	111.0	;
	gDev.sky[	4	].sensor.retractVal	:=	1	;		gDev.sky[	4	].sensor.extendVal	:=	58.2	;
	gDev.sky[	5	].sensor.retractVal	:=	3.2	;		gDev.sky[	5	].sensor.extendVal	:=	106.6	;
	gDev.sky[	6	].sensor.retractVal	:=	6.2	;		gDev.sky[	6	].sensor.extendVal	:=	109.8	;
(*	
	gDev.sky[	7	].sensor.retractVal	:=	1	;		gDev.sky[	7	].sensor.extendVal	:=	113.4	;		//default:115
	gDev.sky[	8	].sensor.retractVal	:=	1	;		gDev.sky[	8	].sensor.extendVal	:=	112.2	;
	gDev.sky[	9	].sensor.retractVal	:=	1	;		gDev.sky[	9	].sensor.extendVal	:=	112.3	;
	gDev.sky[	10	].sensor.retractVal	:=	1	;		gDev.sky[	10	].sensor.extendVal	:=	66.3	;
*)
	
	gDev.sky[	7	].sensor.retractVal	:=	5	;		gDev.sky[	7	].sensor.extendVal	:=	108.7	;		//default:115
	gDev.sky[	8	].sensor.retractVal	:=	8.6	;		gDev.sky[	8	].sensor.extendVal	:=	113.3	;
	gDev.sky[	9	].sensor.retractVal	:=	12.9 ;		gDev.sky[	9	].sensor.extendVal	:=	113.8	;
	gDev.sky[	10	].sensor.retractVal	:=	3.9 ;		gDev.sky[	10	].sensor.extendVal	:=	111.5	;

	
//初始化默认伸缩比例量
	gDev.grd[1].ctrl.exPct :=	28		;			gDev.grd[1].ctrl.rtPct :=	25		;
	gDev.grd[2].ctrl.exPct :=	28		;			gDev.grd[2].ctrl.rtPct :=	25		;
	gDev.grd[3].ctrl.exPct :=	30		;			gDev.grd[3].ctrl.rtPct :=	25		;
	gDev.grd[4].ctrl.exPct :=	28		;			gDev.grd[4].ctrl.rtPct :=	25		;
	gDev.grd[5].ctrl.exPct :=	33		;			gDev.grd[5].ctrl.rtPct :=	33		;		//exPct:=26	rtPct:=21 二次比例
	gDev.grd[6].ctrl.exPct :=	28		;			gDev.grd[6].ctrl.rtPct :=	25		;
	gDev.grd[7].ctrl.exPct :=	28		;			gDev.grd[7].ctrl.rtPct :=	25		;
	gDev.grd[8].ctrl.exPct :=	28		;			gDev.grd[8].ctrl.rtPct :=	25		;
	gDev.grd[9].ctrl.exPct :=	28		;			gDev.grd[9].ctrl.rtPct :=	25		;
	gDev.grd[10].ctrl.exPct :=	28		;			gDev.grd[10].ctrl.rtPct :=	25		;
	
	gDev.sky[0].ctrl.exPct :=	35		;			gDev.sky[0].ctrl.rtPct :=	41		;
	gDev.sky[1].ctrl.exPct :=	25		;			gDev.sky[1].ctrl.rtPct :=	28		;
	gDev.sky[2].ctrl.exPct :=	25		;			gDev.sky[2].ctrl.rtPct :=	28		;
	gDev.sky[3].ctrl.exPct :=	25		;			gDev.sky[3].ctrl.rtPct :=	28		;
	gDev.sky[4].ctrl.exPct :=	25		;			gDev.sky[4].ctrl.rtPct :=	28		;
	gDev.sky[5].ctrl.exPct :=	27		;			gDev.sky[5].ctrl.rtPct :=	30.5	;
	gDev.sky[6].ctrl.exPct :=	25		;			gDev.sky[6].ctrl.rtPct :=	29		;
	gDev.sky[7].ctrl.exPct :=	25		;			gDev.sky[7].ctrl.rtPct :=	28		;
	gDev.sky[8].ctrl.exPct :=	25		;			gDev.sky[8].ctrl.rtPct :=	28		;
	gDev.sky[9].ctrl.exPct :=	25		;			gDev.sky[9].ctrl.rtPct :=	28		;
	gDev.sky[10].ctrl.exPct :=	25		;			gDev.sky[10].ctrl.rtPct :=	28		;



//initialize device name

											gUI.sky[	0	].wname	:=	"天轨1#"	;
gUI.grd[	1	].wname	:=	"地轨1#"	;	gUI.sky[	1	].wname	:=	"天轨2#"	;
gUI.grd[	2	].wname	:=	"地轨2#"	;	gUI.sky[	2	].wname	:=	"天轨3#"	;
gUI.grd[	3	].wname	:=	"地轨3#"	;	gUI.sky[	3	].wname	:=	"天轨4#"	;
gUI.grd[	4	].wname	:=	"地轨4#"	;	gUI.sky[	4	].wname	:=	"天轨5#"	;
gUI.grd[	5	].wname	:=	"地轨5#"	;	gUI.sky[	5	].wname	:=	"天轨6#"	;
gUI.grd[	6	].wname	:=	"地轨6#"	;	gUI.sky[	6	].wname	:=	"天轨7#"	;
gUI.grd[	7	].wname	:=	"地轨7#"	;	gUI.sky[	7	].wname	:=	"天轨8#"	;
gUI.grd[	8	].wname	:=	"地轨8#"	;	gUI.sky[	8	].wname	:=	"天轨9#"	;
gUI.grd[	9	].wname	:=	"地轨9#"	;	gUI.sky[	9	].wname	:=	"天轨10#"	;
gUI.grd[	10	].wname	:=	"地轨10#"	;	gUI.sky[	10	].wname	:=	"天轨11#"	;

												gUI.sky[	0	].hzname	:=	"天.起竖"	;
gUI.grd[	1	].hzname	:=	"地.横1"	;	gUI.sky[	1	].hzname	:=	"天.横1"	;
gUI.grd[	2	].hzname	:=	"地.纵1"	;	gUI.sky[	2	].hzname	:=	"天.纵1"	;
gUI.grd[	3	].hzname	:=	"地.横2"	;	gUI.sky[	3	].hzname	:=	"天.横2"	;
gUI.grd[	4	].hzname	:=	"地.横3"	;	gUI.sky[	4	].hzname	:=	"天.横3"	;
gUI.grd[	5	].hzname	:=	"地.横4"	;	gUI.sky[	5	].hzname	:=	"天.横4"	;
gUI.grd[	6	].hzname	:=	"地.横5"	;	gUI.sky[	6	].hzname	:=	"天.横5"	;
gUI.grd[	7	].hzname	:=	"地.纵2"	;	gUI.sky[	7	].hzname	:=	"天.纵2"	;
gUI.grd[	8	].hzname	:=	"地.横6"	;	gUI.sky[	8	].hzname	:=	"天.横6"	;
gUI.grd[	9	].hzname	:=	"地.横7"	;	gUI.sky[	9	].hzname	:=	"天.横7"	;
gUI.grd[	10	].hzname	:=	"地.横8"	;	gUI.sky[	10	].hzname	:=	"天.横8"	;

											gUI.sky[	0	].name	:=	'SKY_00'	;
gUI.grd[	1	].name	:=	'GRD_01'	;	gUI.sky[	1	].name	:=	'SKY_01'	;
gUI.grd[	2	].name	:=	'GRD_02'	;	gUI.sky[	2	].name	:=	'SKY_02'	;
gUI.grd[	3	].name	:=	'GRD_03'	;	gUI.sky[	3	].name	:=	'SKY_03'	;
gUI.grd[	4	].name	:=	'GRD_04'	;	gUI.sky[	4	].name	:=	'SKY_04'	;
gUI.grd[	5	].name	:=	'GRD_05'	;	gUI.sky[	5	].name	:=	'SKY_05'	;
gUI.grd[	6	].name	:=	'GRD_06'	;	gUI.sky[	6	].name	:=	'SKY_06'	;
gUI.grd[	7	].name	:=	'GRD_07'	;	gUI.sky[	7	].name	:=	'SKY_07'	;
gUI.grd[	8	].name	:=	'GRD_08'	;	gUI.sky[	8	].name	:=	'SKY_08'	;
gUI.grd[	9	].name	:=	'GRD_09'	;	gUI.sky[	9	].name	:=	'SKY_09'	;
gUI.grd[	10	].name	:=	'GRD_10'	;	gUI.sky[	10	].name	:=	'SKY_10'	;



//使用传感器当前位置作为初始化目标位移点
//(*
FOR gi := 1 TO 10 DO
	IF gDev.grd[gi].sensor.position <> 0.0 THEN
		gDev.grd[gi].ctrl.pos.Set_Point := gDev.grd[gi].sensor.position;
	ELSE
		gDev.grd[gi].ctrl.isError := TRUE;
	END_IF
END_FOR

FOR si := 0 TO 10 DO
	IF gDev.sky[si].sensor.position <> 0.0 THEN
		gDev.sky[si].ctrl.pos.Set_Point := gDev.sky[si].sensor.position;
	ELSE
		gDev.sky[si].ctrl.isError := TRUE;
	END_IF
END_FOR
//*)
END_ACTION

ACTION interfaceAct:
//位移值及伸出百分比参数输出	
FOR gi := 1 TO 10 DO
	gUI.grd[gi].postion := gDev.grd[gi].sensor.position;
	gUI.grd[gi].speed := gDev.grd[gi].sensor.speed;
	gUI.grd[gi].extendPercent := percentCalc(1, gi);
END_FOR
FOR si := 0 TO 10 DO
	gUI.sky[si].postion := gDev.sky[si].sensor.position;
	gUI.sky[si].speed := gDev.sky[si].sensor.speed;
	gUI.sky[si].extendPercent := percentCalc(2, si);
END_FOR


//模式判断
pidMode := gUI.mode.usePID;
autoEnableMode := gUI.mode.autoEnable;
autoButtonMode := NOT gUI.mode.manualButtonSet;
autoPctMode := NOT gUI.mode.manualPercentSet;
manualPidPrmSet := gUI.mode.manualSetPid;
//command generetor
FOR gi := 1 TO 10 DO
	IF gUI.grd[gi].btnExtend <> gUI.grd[gi].btnRetract THEN
		gDev.grd[gi].state := DevStatus.runing;
		IF gUI.grd[gi].btnExtend THEN
			gDev.grd[gi].vector := TargetDirect.extend;
			gUI.grd[gi].btnLast := TargetDirect.extend;
		END_IF
		IF gUI.grd[gi].btnRetract THEN
			gDev.grd[gi].vector := TargetDirect.retract;
			gUI.grd[gi].btnLast := TargetDirect.retract;			
		END_IF
	ELSE
		IF gUI.grd[gi].btnExtend THEN
			//伸缩指令不能同时发出，检测到后进行动作转换，重置计数器
			gDev.grd[gi].timeCounter := 0;
			gDev.grd[gi].exeCounter := 0;
			IF gUI.grd[gi].btnLast = TargetDirect.retract THEN
				gDev.grd[gi].vector := TargetDirect.extend;
			ELSE
				gDev.grd[gi].vector := TargetDirect.retract;
			END_IF
			setButtonByDirect(1, gi, gDev.grd[gi].vector);
		ELSE
			gDev.grd[gi].vector := TargetDirect.stop;	
		END_IF
	END_IF
	IF gUI.grd[gi].btnStop THEN
		gDev.grd[gi].vector := TargetDirect.stop;
		setButtonByDirect(1, gi, gDev.grd[gi].vector);
	END_IF
END_FOR

FOR si := 0 TO 10 DO
	IF gUI.sky[si].btnExtend <> gUI.sky[si].btnRetract THEN
		gDev.sky[si].state := DevStatus.runing;
		IF gUI.sky[si].btnExtend THEN
			gDev.sky[si].vector := TargetDirect.extend;
			gUI.sky[si].btnLast := TargetDirect.extend;
		END_IF
		IF gUI.sky[si].btnRetract THEN
			gDev.sky[si].vector := TargetDirect.retract;
			gUI.sky[si].btnLast := TargetDirect.retract;			
		END_IF
	ELSE
		IF gUI.sky[si].btnExtend THEN
			//伸缩指令不能同时发出，检测到后进行动作转换，重置计数器
			gDev.sky[si].timeCounter := 0;
			gDev.sky[si].exeCounter := 0;
			IF gUI.sky[si].btnLast = TargetDirect.retract THEN
				gDev.sky[si].vector := TargetDirect.extend;
			ELSE
				gDev.sky[si].vector := TargetDirect.retract;
			END_IF
			setButtonByDirect(2, si, gDev.sky[si].vector);
		ELSE
			gDev.sky[si].vector := TargetDirect.stop;
		END_IF
	END_IF
	IF gUI.sky[si].btnStop THEN
		gDev.sky[si].vector := TargetDirect.stop;
		setButtonByDirect(1, gi, gDev.grd[gi].vector);
	END_IF
END_FOR
END_ACTION

ACTION autoResetButton:

//更新Button
FOR gi := 1 TO 10 DO
	setButtonByDirect(1, gi, gDev.grd[gi].vector);
END_FOR


FOR si := 0 TO 10 DO
	setButtonByDirect(2, si, gDev.sky[si].vector);
END_FOR
END_ACTION

METHOD manualExecute
VAR_INPUT
END_VAR
VAR
	//targetDirect		:TargetDirect;
END_VAR
FOR gi := 1 TO 10 DO
	IF gUI.grd[gi].pwrEnable THEN
		cmdExecutor0(level := 1, idx := gi, 
					direct := gDev.grd[gi].vector, 
					percent := gUI.grd[gi].pwrPercent);
	ELSE
		cmdExecutor0(level := 1, idx := gi, direct := 3, percent := 0);		
	END_IF
END_FOR

FOR si := 0 TO 10 DO
	IF gUI.sky[si].pwrEnable THEN
		cmdExecutor0(level := 2, idx := si, 
					direct := gDev.sky[si].vector, 
					percent := gUI.sky[si].pwrPercent);	
	ELSE
		cmdExecutor0(level := 2, idx := si, direct := 3, percent := 0);		
	END_IF
END_FOR
END_METHOD

METHOD pidExecute
VAR_INPUT
END_VAR
VAR
	vector 		:TargetDirect;
END_VAR
FOR gi := 1 TO 10 DO
	IF gDev.grd[gi].ctrl.isError THEN
		CONTINUE;
	END_IF
	cmdExecutor(level := 1, idx := gi, percent := grdPid[gi].res);
END_FOR


FOR si := 1 TO 10 DO
	IF gDev.sky[si].ctrl.isError THEN
		CONTINUE;
	END_IF
	cmdExecutor(level := 2, idx := si, percent := skyPid[si].res);
END_FOR

//起竖挡板执行开关量
IF NOT gDev.sky[0].ctrl.isError THEN
	IF gDev.sky[0].vector = TargetDirect.extend THEN
		cmdExecutor(level := 2, idx := 0, percent := gDev.sky[0].ctrl.exPct);
	END_IF
	IF gDev.sky[0].vector = TargetDirect.retract THEN
		cmdExecutor(level := 2, idx := 0, percent := -gDev.sky[0].ctrl.rtPct);
	END_IF
END_IF
(*
IF NOT gDev.grd[7].ctrl.isError THEN
	IF gDev.grd[7].vector = TargetDirect.extend THEN
		cmdExecutor(level := 1, idx := 7, percent := gDev.grd[7].ctrl.exPct);
	END_IF
	IF gDev.grd[7].vector = TargetDirect.retract THEN
		cmdExecutor(level := 1, idx := 7, percent := -gDev.grd[7].ctrl.rtPct);
	END_IF
END_IF	
IF NOT gDev.sky[7].ctrl.isError THEN
	IF gDev.sky[7].vector = TargetDirect.extend THEN
		cmdExecutor(level := 2, idx := 7, percent := gDev.sky[7].ctrl.exPct);
	END_IF
	IF gDev.sky[7].vector = TargetDirect.retract THEN
		cmdExecutor(level := 2, idx := 7, percent := -gDev.sky[7].ctrl.rtPct);
	END_IF
END_IF
*)
END_METHOD

METHOD pidTestUi
VAR_INPUT
END_VAR

VAR

END_VAR
IF gUI.pid.level = 1 AND gUI.pid.idx = 0 THEN	//地轨从1-10，天轨从0-10
	RETURN;
END_IF

IF gUI.mode.syncExt THEN
	gUI.grd[gUI.pid.idx].btnExtend := TRUE;gUI.sky[gUI.pid.idx].btnExtend := TRUE;
END_IF
IF gUI.mode.syncRct THEN
	gUI.grd[gUI.pid.idx].btnRetract := TRUE;gUI.sky[gUI.pid.idx].btnRetract := TRUE;
END_IF


IF (NOT gUI.pid.posBtn) THEN
	RETURN;
END_IF

IF gUI.pid.level = 1 THEN 	//地轨部分
	IF idx = gUI.pid.idx THEN		//标号相同更新设备参数
		
		gUI.pid.devSetPos := gDev.grd[idx].ctrl.pos.Set_Point;
		gUI.pid.executeVal := grdPid[idx].res;
		resetPidParam := gUI.pid.rstPidBtn;
		//-----------------位置环------------------------------//
		gUI.pid.pos.Act_Val := gDev.grd[idx].sensor.position;
		gUI.pid.pos.Err := gUI.pid.pos.Set_Point - gUI.pid.pos.Act_Val;
		gUI.pid.pos.OUT := gDev.grd[idx].ctrl.pos.OUT;
		gDev.grd[idx].ctrl.pos := gUI.pid.pos;
		//-----------------速度环------------------------------//
		gUI.pid.spd.Act_Val := gDev.grd[idx].sensor.speed;
		gUI.pid.spd.Err := gUI.pid.spd.Set_Point - gUI.pid.spd.Act_Val;
		gUI.pid.spd.OUT := gDev.sky[idx].ctrl.spd.OUT;
		gDev.grd[idx].ctrl.spd := gUI.pid.spd;
		//-----------------前馈参数------------------------------//
		gDev.grd[idx].ctrl.ff := gUI.pid.ff;	
		
	ELSE							//标号不同，更新界面参数
		idx := gUI.pid.idx;
		gUI.pid.pos := gDev.grd[idx].ctrl.pos;
		gUI.pid.spd := gDev.grd[idx].ctrl.spd;
		gUI.pid.ff	:= gDev.grd[idx].ctrl.ff;	
	END_IF			
END_IF
IF gUI.pid.level = 2 THEN 					//天轨部分
	IF idx = gUI.pid.idx THEN		//标号相同更新设备参数
		
		//-----------------位置环------------------------------//
		gUI.pid.pos.Act_Val := gDev.sky[idx].sensor.position;
		gUI.pid.pos.Err := gUI.pid.pos.Set_Point - gUI.pid.pos.Act_Val;
		gUI.pid.pos.OUT := gDev.sky[idx].ctrl.pos.OUT;
		gDev.sky[idx].ctrl.pos := gUI.pid.pos;
		//-----------------速度环------------------------------//
		gUI.pid.spd.Act_Val := gDev.sky[idx].sensor.speed;
		gUI.pid.spd.Err := gUI.pid.spd.Set_Point - gUI.pid.spd.Act_Val;
		gUI.pid.spd.OUT := gDev.sky[idx].ctrl.spd.OUT;
		gDev.sky[idx].ctrl.spd := gUI.pid.spd;
		//-----------------前馈参数------------------------------//
		gDev.sky[idx].ctrl.ff := gUI.pid.ff;	

		gUI.pid.devSetPos := gDev.sky[idx].ctrl.pos.Set_Point;
		gUI.pid.executeVal := skyPid[idx].res;
		resetPidParam := gUI.pid.rstPidBtn;

	ELSE							//标号不同，更新界面参数
		idx := gUI.pid.idx;
		gUI.pid.pos := gDev.sky[idx].ctrl.pos;
		gUI.pid.spd := gDev.sky[idx].ctrl.spd;
		gUI.pid.ff	:= gDev.sky[idx].ctrl.ff;

	END_IF			

END_IF
END_METHOD

ACTION autoEnable:

IF pidMode THEN 	//pid模式，没有动作指令时不执行输出
	
	IF NOT manualPidPrmSet THEN
		FOR gi := 1 TO 10 DO
			 IF gDev.grd[gi].vector = TargetDirect.stop THEN
				cmdExecutor(level := 1, idx := gi, percent := 0);
			 END_IF
		END_FOR
		
		FOR si := 1 TO 10 DO
			IF gDev.sky[si].vector = TargetDirect.stop THEN		
				cmdExecutor(level := 2, idx := si, percent := 0);
			END_IF
		END_FOR
		//起竖挡板执行开关量特判
		IF gDev.sky[0].vector = TargetDirect.stop THEN 
			cmdExecutor(level := 2, idx := 0, percent := 0);
		END_IF
	END_IF
ELSE		//开关量控制
	
	FOR gi := 1 TO 10 DO
		 IF gDev.grd[gi].vector = TargetDirect.stop THEN
			gUI.grd[gi].pwrEnable := FALSE;
		 ELSE
			gUI.grd[gi].pwrEnable := TRUE;
		 END_IF
	END_FOR
	
	FOR si := 0 TO 10 DO
		IF gDev.sky[si].vector = TargetDirect.stop THEN		
			gUI.sky[si].pwrEnable := FALSE;
		ELSE													
			gUI.sky[si].pwrEnable := TRUE;	
		END_IF
	END_FOR
END_IF

(*
FOR gi := 1 TO 10 DO
	 IF gDev.grd[gi].vector <> TargetDirect.stop THEN
		IF pidMode THEN
			cmdExecutor(level := 1, idx := gi, percent := grdPid[gi].res);
		ELSE
			gUI.grd[gi].pwrEnable := TRUE;
		END_IF
	 ELSE
		IF pidMode THEN
			cmdExecutor(level := 1, idx := gi, percent := 0);
		ELSE
			gUI.grd[gi].pwrEnable := FALSE;
		END_IF
	 END_IF
END_FOR


FOR si := 1 TO 10 DO
	IF gDev.sky[si].vector <> TargetDirect.stop THEN		//运动状态，执行  PID或开关使能
		IF pidMode THEN
			cmdExecutor(level := 2, idx := si, percent := skyPid[si].res);
		ELSE
			gUI.sky[si].pwrEnable := TRUE;	
		END_IF
	ELSE													//停止状态，关闭 PID或开关使能
		IF pidMode THEN
			cmdExecutor(level := 2, idx := si, percent := 0);
		ELSE
			gUI.sky[si].pwrEnable := FALSE;
		END_IF
	END_IF
END_FOR

IF gDev.sky[0].vector <> TargetDirect.stop THEN
	gUI.sky[0].pwrEnable := TRUE;
	IF gDev.sky[0].vector = TargetDirect.extend THEN	cmdExecutor(level := 2, idx := 0, percent := gDev.sky[0].ctrl.exPct);END_IF
	IF gDev.sky[0].vector = TargetDirect.retract THEN	cmdExecutor(level := 2, idx := 0, percent := -gDev.sky[0].ctrl.rtPct);END_IF
ELSE
	gUI.sky[0].pwrEnable := FALSE;
	cmdExecutor(level := 2, idx := 0, percent := 0);
END_IF
*)
END_ACTION

METHOD pidCalc
VAR_INPUT
END_VAR
VAR
	vector			:TargetDirect;
END_VAR
FOR gi := 1 TO 10 DO
	IF NOT manualPidPrmSet THEN
		vector := gDev.grd[gi].vector;
		CASE vector OF
			TargetDirect.stop:
			CASE gDev.grd[gi].state OF
				DevStatus.extended:
					gDev.grd[gi].ctrl.pos.Set_Point := gDev.grd[gi].ctrl.extVal;
				DevStatus.retracted:
					gDev.grd[gi].ctrl.pos.Set_Point := gDev.grd[gi].ctrl.rtcVal;
				ELSE
					gDev.grd[gi].ctrl.pos.Set_Point := gDev.grd[gi].sensor.position;
			END_CASE			
			TargetDirect.extend:
				gDev.grd[gi].ctrl.pos.Set_Point := gDev.grd[gi].ctrl.extVal;
			TargetDirect.retract:
				gDev.grd[gi].ctrl.pos.Set_Point := gDev.grd[gi].ctrl.rtcVal;
		END_CASE
END_IF
	
	grdPid[gi](idx := gi, isReset := resetPidParam, cycTimer := 0.01, res => );

END_FOR

FOR si := 0 TO 10 DO
	IF NOT manualPidPrmSet THEN
		vector := gDev.sky[si].vector;
		CASE vector OF
			TargetDirect.stop:
			CASE gDev.sky[si].state OF
				DevStatus.extended:
					gDev.sky[si].ctrl.pos.Set_Point := gDev.sky[si].ctrl.extVal;
				DevStatus.retracted:
					gDev.sky[si].ctrl.pos.Set_Point := gDev.sky[si].ctrl.rtcVal;
				ELSE
					gDev.sky[si].ctrl.pos.Set_Point := gDev.sky[si].sensor.position;
			END_CASE			
			TargetDirect.extend:
				gDev.sky[si].ctrl.pos.Set_Point := gDev.sky[si].ctrl.extVal;
			TargetDirect.retract:
				gDev.sky[si].ctrl.pos.Set_Point := gDev.sky[si].ctrl.rtcVal;
		END_CASE
		
		
	END_IF
	skyPid[si](idx := si, isReset := resetPidParam, cycTimer := 0.01, res =>);
END_FOR
END_METHOD

ACTION setExecutePercent:
FOR gi := 1 TO 10 DO
	IF gUI.grd[gi].btnExtend THEN
		gUI.grd[gi].pwrPercent := gDev.grd[gi].ctrl.exPct;
	END_IF
	IF gUI.grd[gi].btnRetract THEN
		gUI.grd[gi].pwrPercent := gDev.grd[gi].ctrl.rtPct;
	END_IF
END_FOR

FOR si := 0 TO 10 DO
	IF gUI.sky[si].btnExtend THEN
		gUI.sky[si].pwrPercent := gDev.sky[si].ctrl.exPct;
	END_IF
	IF gUI.sky[si].btnRetract THEN
		gUI.sky[si].pwrPercent := gDev.sky[si].ctrl.rtPct;
	END_IF
END_FOR

//grd[5]比例输出特判(延时时间过长，小信号无法动作，动作后速度过快的问题)使用速度传感器判定
IF gUI.grd[5].btnExtend THEN 
	IF ABS(gDev.grd[5].sensor.extendVal - gDev.grd[5].sensor.position) < 25 THEN
		gUI.grd[5].pwrPercent := 22;	
	END_IF
END_IF
IF gUI.grd[5].btnRetract THEN 
	IF ABS(gDev.grd[5].sensor.retractVal - gDev.grd[5].sensor.position) < 30 THEN
		gUI.grd[5].pwrPercent := 22;	
	END_IF
END_IF

//其他特判
(*IF gUI.grd[2].btnRetract THEN 
	IF ABS(gDev.grd[2].sensor.retractVal - gDev.grd[2].sensor.position) < 20 THEN
		gUI.grd[2].pwrPercent := 21;	
	END_IF
END_IF*)
IF gUI.grd[6].btnRetract THEN 
	IF ABS(gDev.grd[6].sensor.retractVal - gDev.grd[6].sensor.position) < 25 THEN
		gUI.grd[6].pwrPercent := 21;	
	END_IF
END_IF
END_ACTION

ACTION initializePid:

//PID param
gDev.grd[	1	].ctrl.pos.Kp	:=	1.2	;	gDev.grd[	1	].ctrl.spd.Kp	:=	0.05	;
gDev.grd[	1	].ctrl.pos.Ki	:=	0	;	gDev.grd[	1	].ctrl.spd.Ki	:=	0		;
gDev.grd[	1	].ctrl.pos.Kd	:=	0	;	gDev.grd[	1	].ctrl.spd.Kd	:=	0.02	;
											
gDev.grd[	2	].ctrl.pos.Kp	:=	1.3	;	gDev.grd[	2	].ctrl.spd.Kp	:=	0.05	;
gDev.grd[	2	].ctrl.pos.Ki	:=	0	;	gDev.grd[	2	].ctrl.spd.Ki	:=	0		;
gDev.grd[	2	].ctrl.pos.Kd	:=	0	;	gDev.grd[	2	].ctrl.spd.Kd	:=	0.002	;
gDev.grd[	3	].ctrl.pos.Kp	:=	1	;	gDev.grd[	3	].ctrl.spd.Kp	:=	0.01	;
gDev.grd[	3	].ctrl.pos.Ki	:=	0	;	gDev.grd[	3	].ctrl.spd.Ki	:=	0		;
gDev.grd[	3	].ctrl.pos.Kd	:=	0	;	gDev.grd[	3	].ctrl.spd.Kd	:=	0		;
											
gDev.grd[	4	].ctrl.pos.Kp	:=	0	;	gDev.grd[	4	].ctrl.spd.Kp	:=	0		;
gDev.grd[	4	].ctrl.pos.Ki	:=	0	;	gDev.grd[	4	].ctrl.spd.Ki	:=	0		;
gDev.grd[	4	].ctrl.pos.Kd	:=	0	;	gDev.grd[	4	].ctrl.spd.Kd	:=	0		;
gDev.grd[	5	].ctrl.pos.Kp	:=	1.2	;	gDev.grd[	5	].ctrl.spd.Kp	:=	0.01	;
gDev.grd[	5	].ctrl.pos.Ki	:=	0	;	gDev.grd[	5	].ctrl.spd.Ki	:=	0		;
gDev.grd[	5	].ctrl.pos.Kd	:=	0	;	gDev.grd[	5	].ctrl.spd.Kd	:=	0		;
											
gDev.grd[	6	].ctrl.pos.Kp	:=	1.2	;	gDev.grd[	6	].ctrl.spd.Kp	:=	0.01	;
gDev.grd[	6	].ctrl.pos.Ki	:=	0	;	gDev.grd[	6	].ctrl.spd.Ki	:=	0		;
gDev.grd[	6	].ctrl.pos.Kd	:=	0	;	gDev.grd[	6	].ctrl.spd.Kd	:=	0		;
gDev.grd[	7	].ctrl.pos.Kp	:=	1.1	;	gDev.grd[	7	].ctrl.spd.Kp	:=	0.02		;
gDev.grd[	7	].ctrl.pos.Ki	:=	0	;	gDev.grd[	7	].ctrl.spd.Ki	:=	0		;
gDev.grd[	7	].ctrl.pos.Kd	:=	0	;	gDev.grd[	7	].ctrl.spd.Kd	:=	0		;
											
gDev.grd[	8	].ctrl.pos.Kp	:=	1.1	;	gDev.grd[	8	].ctrl.spd.Kp	:=	0.01		;
gDev.grd[	8	].ctrl.pos.Ki	:=	0	;	gDev.grd[	8	].ctrl.spd.Ki	:=	0		;
gDev.grd[	8	].ctrl.pos.Kd	:=	0	;	gDev.grd[	8	].ctrl.spd.Kd	:=	0		;
gDev.grd[	9	].ctrl.pos.Kp	:=	1.1	;	gDev.grd[	9	].ctrl.spd.Kp	:=	0.05		;
gDev.grd[	9	].ctrl.pos.Ki	:=	0	;	gDev.grd[	9	].ctrl.spd.Ki	:=	0		;
gDev.grd[	9	].ctrl.pos.Kd	:=	0	;	gDev.grd[	9	].ctrl.spd.Kd	:=	0		;
gDev.grd[	10	].ctrl.pos.Kp	:=	1.1	;	gDev.grd[	10	].ctrl.spd.Kp	:=	0.02		;
gDev.grd[	10	].ctrl.pos.Ki	:=	0	;	gDev.grd[	10	].ctrl.spd.Ki	:=	0		;
gDev.grd[	10	].ctrl.pos.Kd	:=	0	;	gDev.grd[	10	].ctrl.spd.Kd	:=	0		;
											
											
											
gDev.sky[	0	].ctrl.pos.Kp	:=	1.0	;	gDev.sky[	0	].ctrl.spd.Kp	:=	0.01	;
gDev.sky[	0	].ctrl.pos.Ki	:=	0	;	gDev.sky[	0	].ctrl.spd.Ki	:=	0		;
gDev.sky[	0	].ctrl.pos.Kd	:=	0.1	;	gDev.sky[	0	].ctrl.spd.Kd	:=	0.001	;
gDev.sky[	1	].ctrl.pos.Kp	:=	1.0	;	gDev.sky[	1	].ctrl.spd.Kp	:=	0.01	;
gDev.sky[	1	].ctrl.pos.Ki	:=	0	;	gDev.sky[	1	].ctrl.spd.Ki	:=	0		;
gDev.sky[	1	].ctrl.pos.Kd	:=	0	;	gDev.sky[	1	].ctrl.spd.Kd	:=	0.001	;
											
gDev.sky[	2	].ctrl.pos.Kp	:=	1.1	;	gDev.sky[	2	].ctrl.spd.Kp	:=	0.02	;
gDev.sky[	2	].ctrl.pos.Ki	:=	0	;	gDev.sky[	2	].ctrl.spd.Ki	:=	0		;
gDev.sky[	2	].ctrl.pos.Kd	:=	0	;	gDev.sky[	2	].ctrl.spd.Kd	:=	0.001	;
gDev.sky[	3	].ctrl.pos.Kp	:=	1.1	;	gDev.sky[	3	].ctrl.spd.Kp	:=	0.02	;
gDev.sky[	3	].ctrl.pos.Ki	:=	0	;	gDev.sky[	3	].ctrl.spd.Ki	:=	0		;
gDev.sky[	3	].ctrl.pos.Kd	:=	0.02;	gDev.sky[	3	].ctrl.spd.Kd	:=	0.001	;
											
gDev.sky[	4	].ctrl.pos.Kp	:=	0	;	gDev.sky[	4	].ctrl.spd.Kp	:=	0		;
gDev.sky[	4	].ctrl.pos.Ki	:=	0	;	gDev.sky[	4	].ctrl.spd.Ki	:=	0		;
gDev.sky[	4	].ctrl.pos.Kd	:=	0	;	gDev.sky[	4	].ctrl.spd.Kd	:=	0		;
gDev.sky[	5	].ctrl.pos.Kp	:=	1.2	;	gDev.sky[	5	].ctrl.spd.Kp	:=	0.01	;
gDev.sky[	5	].ctrl.pos.Ki	:=	0	;	gDev.sky[	5	].ctrl.spd.Ki	:=	0		;
gDev.sky[	5	].ctrl.pos.Kd	:=	0	;	gDev.sky[	5	].ctrl.spd.Kd	:=	0.001	;
											
gDev.sky[	6	].ctrl.pos.Kp	:=	1.1	;	gDev.sky[	6	].ctrl.spd.Kp	:=	0.01	;
gDev.sky[	6	].ctrl.pos.Ki	:=	0	;	gDev.sky[	6	].ctrl.spd.Ki	:=	0		;
gDev.sky[	6	].ctrl.pos.Kd	:=	0.01;	gDev.sky[	6	].ctrl.spd.Kd	:=	0.001	;
gDev.sky[	7	].ctrl.pos.Kp	:=	1.1	;	gDev.sky[	7	].ctrl.spd.Kp	:=	0.01	;
gDev.sky[	7	].ctrl.pos.Ki	:=	0	;	gDev.sky[	7	].ctrl.spd.Ki	:=	0		;
gDev.sky[	7	].ctrl.pos.Kd	:=	0	;	gDev.sky[	7	].ctrl.spd.Kd	:=	0		;
											
gDev.sky[	8	].ctrl.pos.Kp	:=	1.1	;	gDev.sky[	8	].ctrl.spd.Kp	:=	0.01	;
gDev.sky[	8	].ctrl.pos.Ki	:=	0	;	gDev.sky[	8	].ctrl.spd.Ki	:=	0		;
gDev.sky[	8	].ctrl.pos.Kd	:=	0	;	gDev.sky[	8	].ctrl.spd.Kd	:=	0		;
gDev.sky[	9	].ctrl.pos.Kp	:=	1.2	;	gDev.sky[	9	].ctrl.spd.Kp	:=	0.01		;
gDev.sky[	9	].ctrl.pos.Ki	:=	0	;	gDev.sky[	9	].ctrl.spd.Ki	:=	0		;
gDev.sky[	9	].ctrl.pos.Kd	:=	0	;	gDev.sky[	9	].ctrl.spd.Kd	:=	0		;
gDev.sky[	10	].ctrl.pos.Kp	:=	1.1	;	gDev.sky[	10	].ctrl.spd.Kp	:=	0		;
gDev.sky[	10	].ctrl.pos.Ki	:=	0	;	gDev.sky[	10	].ctrl.spd.Ki	:=	0		;
gDev.sky[	10	].ctrl.pos.Kd	:=	0	;	gDev.sky[	10	].ctrl.spd.Kd	:=	0		;


gDev.grd[1	].ctrl.ff.pstThreshold	:=	18.5	;	gDev.grd[1	].ctrl.ff.pstKv	:=	0.35 	;	
gDev.grd[1	].ctrl.ff.negThreshold	:=	15  	;	gDev.grd[1	].ctrl.ff.negKv	:=	0.27	;
gDev.grd[2	].ctrl.ff.pstThreshold	:=	18  	;	gDev.grd[2	].ctrl.ff.pstKv	:=	0.27	;	
gDev.grd[2	].ctrl.ff.negThreshold	:=	16  	;	gDev.grd[2	].ctrl.ff.negKv	:=	0.27	;
gDev.grd[3	].ctrl.ff.pstThreshold	:=	19  	;	gDev.grd[3	].ctrl.ff.pstKv	:=	0.3 	;	
gDev.grd[3	].ctrl.ff.negThreshold	:=	16  	;	gDev.grd[3	].ctrl.ff.negKv	:=	0.3 	;
gDev.grd[4	].ctrl.ff.pstThreshold	:=	0   	;	gDev.grd[4	].ctrl.ff.pstKv	:=	0   	;	
gDev.grd[4	].ctrl.ff.negThreshold	:=	0   	;	gDev.grd[4	].ctrl.ff.negKv	:=	0   	;
gDev.grd[5	].ctrl.ff.pstThreshold	:=	18  	;	gDev.grd[5	].ctrl.ff.pstKv	:=	0.3 	;	
gDev.grd[5	].ctrl.ff.negThreshold	:=	17  	;	gDev.grd[5	].ctrl.ff.negKv	:=	0.3 	;
gDev.grd[6	].ctrl.ff.pstThreshold	:=	18.5	;	gDev.grd[6	].ctrl.ff.pstKv	:=	0.28	;	
gDev.grd[6	].ctrl.ff.negThreshold	:=	17  	;	gDev.grd[6	].ctrl.ff.negKv	:=	0.28	;
gDev.grd[7	].ctrl.ff.pstThreshold	:=	17   	;	gDev.grd[7	].ctrl.ff.pstKv	:=	0.36  	;	
gDev.grd[7	].ctrl.ff.negThreshold	:=	15   	;	gDev.grd[7	].ctrl.ff.negKv	:=	0.29  	;
gDev.grd[8	].ctrl.ff.pstThreshold	:=	19   	;	gDev.grd[8	].ctrl.ff.pstKv	:=	0.4   	;	
gDev.grd[8	].ctrl.ff.negThreshold	:=	17  	;	gDev.grd[8	].ctrl.ff.negKv	:=	0.3   	;
gDev.grd[9	].ctrl.ff.pstThreshold	:=	18   	;	gDev.grd[9	].ctrl.ff.pstKv	:=	0.45   	;	
gDev.grd[9	].ctrl.ff.negThreshold	:=	17   	;	gDev.grd[9	].ctrl.ff.negKv	:=	0.28  	;
gDev.grd[10	].ctrl.ff.pstThreshold	:=	19   	;	gDev.grd[10	].ctrl.ff.pstKv	:=	0.30   	;	
gDev.grd[10	].ctrl.ff.negThreshold	:=	19.5   	;	gDev.grd[10	].ctrl.ff.negKv	:=	0.25   	;

gDev.sky[0	].ctrl.ff.pstThreshold	:=	22		;	gDev.sky[0	].ctrl.ff.pstKv	:=	0.29	;	
gDev.sky[0	].ctrl.ff.negThreshold	:=	18		;	gDev.sky[0	].ctrl.ff.negKv	:=	0.25	;
gDev.sky[1	].ctrl.ff.pstThreshold	:=	14.8	;	gDev.sky[1	].ctrl.ff.pstKv	:=	0.4 	;	
gDev.sky[1	].ctrl.ff.negThreshold	:=	18.5	;	gDev.sky[1	].ctrl.ff.negKv	:=	0.32	;
gDev.sky[2	].ctrl.ff.pstThreshold	:=	17.5	;	gDev.sky[2	].ctrl.ff.pstKv	:=	0.33	;	
gDev.sky[2	].ctrl.ff.negThreshold	:=	18.3	;	gDev.sky[2	].ctrl.ff.negKv	:=	0.26	;
gDev.sky[3	].ctrl.ff.pstThreshold	:=	17.8	;	gDev.sky[3	].ctrl.ff.pstKv	:=	0.37	;	
gDev.sky[3	].ctrl.ff.negThreshold	:=	17.5	;	gDev.sky[3	].ctrl.ff.negKv	:=	0.33	;
gDev.sky[4	].ctrl.ff.pstThreshold	:=	0		;	gDev.sky[4	].ctrl.ff.pstKv	:=	0		;	
gDev.sky[4	].ctrl.ff.negThreshold	:=	0		;	gDev.sky[4	].ctrl.ff.negKv	:=	0		;
gDev.sky[5	].ctrl.ff.pstThreshold	:=	18.0	;	gDev.sky[5	].ctrl.ff.pstKv	:=	0.30	;	
gDev.sky[5	].ctrl.ff.negThreshold	:=	28.5	;	gDev.sky[5	].ctrl.ff.negKv	:=	0.40	;
gDev.sky[6	].ctrl.ff.pstThreshold	:=	16.8	;	gDev.sky[6	].ctrl.ff.pstKv	:=	0.35	;	
gDev.sky[6	].ctrl.ff.negThreshold	:=	18.8	;	gDev.sky[6	].ctrl.ff.negKv	:=	0.29	;
gDev.sky[7	].ctrl.ff.pstThreshold	:=	17.5	;	gDev.sky[7	].ctrl.ff.pstKv	:=	0.32	;	
gDev.sky[7	].ctrl.ff.negThreshold	:=	18.5	;	gDev.sky[7	].ctrl.ff.negKv	:=	0.30	;
gDev.sky[8	].ctrl.ff.pstThreshold	:=	18		;	gDev.sky[8	].ctrl.ff.pstKv	:=	0.3		;	
gDev.sky[8	].ctrl.ff.negThreshold	:=	20.5	;	gDev.sky[8	].ctrl.ff.negKv	:=	0.25	;
gDev.sky[9	].ctrl.ff.pstThreshold	:=	15.5	;	gDev.sky[9	].ctrl.ff.pstKv	:=	0.38	;	
gDev.sky[9	].ctrl.ff.negThreshold	:=	17.0	;	gDev.sky[9	].ctrl.ff.negKv	:=	0.27	;
gDev.sky[10	].ctrl.ff.pstThreshold	:=	17		;	gDev.sky[10	].ctrl.ff.pstKv	:=	0.32	;	
gDev.sky[10	].ctrl.ff.negThreshold	:=	17  	;	gDev.sky[10	].ctrl.ff.negKv	:=	0.3		;



//更新pid伸缩设定位置
FOR gi := 1 TO 10 DO
	gDev.grd[gi].ctrl.extVal := gDev.grd[gi].sensor.extendVal;
	gDev.grd[gi].ctrl.rtcVal := gDev.grd[gi].sensor.retractVal;
END_FOR

FOR si := 0 TO 10 DO
	gDev.sky[si].ctrl.extVal := gDev.sky[si].sensor.extendVal;
	gDev.sky[si].ctrl.rtcVal := gDev.sky[si].sensor.retractVal;
END_FOR
//天地轨伸出均可白嫖位移值,缩回动作不行
gDev.grd[1].ctrl.extVal := gDev.grd[1].sensor.extendVal + 4;
gDev.grd[1].ctrl.rtcVal := gDev.grd[1].sensor.retractVal - 5.4;
gDev.grd[2].ctrl.rtcVal := gDev.grd[2].sensor.retractVal - 5.4;
gDev.grd[2].ctrl.extVal := gDev.grd[2].sensor.extendVal + 3;
gDev.grd[3].ctrl.extVal := gDev.grd[3].sensor.extendVal + 6;
gDev.grd[3].ctrl.rtcVal := gDev.grd[3].sensor.retractVal - 10.5;
gDev.grd[5].ctrl.extVal := gDev.grd[5].sensor.extendVal + 2.5;
gDev.grd[5].ctrl.rtcVal := gDev.grd[5].sensor.retractVal - 1.2-2;
gDev.grd[6].ctrl.extVal := gDev.grd[6].sensor.extendVal + 5.5;
gDev.grd[6].ctrl.rtcVal := gDev.grd[6].sensor.retractVal - 5.5;
gDev.grd[7].ctrl.extVal := gDev.grd[7].sensor.extendVal + 5.3;
gDev.grd[7].ctrl.rtcVal := gDev.grd[7].sensor.retractVal - 15;
gDev.grd[8].ctrl.extVal := gDev.grd[8].sensor.extendVal + 7.1;
gDev.grd[8].ctrl.rtcVal := gDev.grd[8].sensor.retractVal - 16.5;
gDev.grd[9].ctrl.extVal := gDev.grd[9].sensor.extendVal + 4  ;
gDev.grd[9].ctrl.rtcVal := gDev.grd[9].sensor.retractVal - 4 ;

gDev.sky[0].ctrl.rtcVal := gDev.sky[0].sensor.retractVal - 9.0;		//2.7
gDev.sky[1].ctrl.extVal := gDev.sky[1].sensor.extendVal + 7;
gDev.sky[1].ctrl.rtcVal := gDev.sky[1].sensor.retractVal - 6.8;
gDev.sky[2].ctrl.extVal := gDev.sky[2].sensor.extendVal + 2;
gDev.sky[2].ctrl.rtcVal := gDev.sky[2].sensor.retractVal - 3.5;
gDev.sky[3].ctrl.extVal := gDev.sky[3].sensor.extendVal + 7.5;
gDev.sky[3].ctrl.rtcVal := gDev.sky[3].sensor.retractVal - 8.5;
gDev.sky[5].ctrl.extVal := gDev.sky[5].sensor.extendVal + 8 ;
gDev.sky[5].ctrl.rtcVal := gDev.sky[5].sensor.retractVal - 13;
gDev.sky[6].ctrl.extVal := gDev.sky[6].sensor.extendVal + 6;
gDev.sky[6].ctrl.rtcVal := gDev.sky[6].sensor.retractVal - 6;
gDev.sky[7].ctrl.extVal := gDev.sky[7].sensor.extendVal + 5;
gDev.sky[7].ctrl.rtcVal := gDev.sky[7].sensor.retractVal - 4.2;
gDev.sky[9].ctrl.extVal := gDev.sky[9].sensor.extendVal + 2.2;
gDev.sky[9].ctrl.rtcVal := gDev.sky[9].sensor.retractVal - 11;
gDev.sky[10].ctrl.extVal := gDev.sky[10].sensor.extendVal + 9;
gDev.sky[10].ctrl.rtcVal := gDev.sky[10].sensor.retractVal - 11;



FOR gi := 1 TO 10 DO
	gDev.grd[	gi	].ctrl.pos.Max_Val	:=	60	;
	gDev.grd[	gi	].ctrl.pos.Max_ACC	:=	120	;
	gDev.grd[	gi	].ctrl.spd.Max_Val	:=	40	;
	gDev.grd[	gi	].ctrl.spd.Max_ACC	:=	150	;
END_FOR

FOR si := 0 TO 10 DO
	gDev.sky[	si	].ctrl.pos.Max_Val	:=	60	;
	gDev.sky[	si	].ctrl.pos.Max_ACC	:=	120	;
	gDev.sky[	si	].ctrl.spd.Max_Val	:=	40	;
	gDev.sky[	si	].ctrl.spd.Max_ACC	:=	150	;
END_FOR
END_ACTION

END_PROGRAM

// Device/Application/basefun/CommandExecutor0
FUNCTION_BLOCK CommandExecutor0
VAR_INPUT
	level		:INT;			//1->地轨	2->天轨
	idx			:INT;			//挡板索引编号
	direct		:TargetDirect;	//方向
	percent		:REAL;			//比例阀百分比 传入0-100
END_VAR
VAR_OUTPUT
END_VAR
VAR
END_VAR


CASE direct OF
	TargetDirect.extend:
		CASE level OF
			1:
				gController.grd[idx].extendPercent := REAL_TO_WORD(percent * 65535 / 100);
				gController.grd[idx].retractPercent := 0;
			2:
				gController.sky[idx].extendPercent := REAL_TO_WORD(percent * 65535 / 100);
				gController.sky[idx].retractPercent := 0;
		END_CASE
	TargetDirect.retract:
		CASE level OF
			1:
				gController.grd[idx].extendPercent := 0;
				gController.grd[idx].retractPercent := REAL_TO_WORD(percent * 65535 / 100);
			2:
				gController.sky[idx].extendPercent := 0;
				gController.sky[idx].retractPercent := REAL_TO_WORD(percent * 65535 / 100);
		END_CASE
	TargetDirect.stop:
		CASE level OF
			1:
				gController.grd[idx].extendPercent := 0;
				gController.grd[idx].retractPercent := 0;
			2:
				gController.sky[idx].extendPercent := 0;
				gController.sky[idx].retractPercent := 0;
		END_CASE
	
	ELSE
		CASE level OF
			1:
				gController.grd[idx].extendPercent := 0;
				gController.grd[idx].retractPercent := 0;
			2:
				gController.sky[idx].extendPercent := 0;
				gController.sky[idx].retractPercent := 0;
		END_CASE
		
END_CASE

END_FUNCTION_BLOCK

// Device/Application/basefun/CommandExecutor

FUNCTION_BLOCK CommandExecutor
VAR_INPUT
	level		:INT;			//1->地轨	2->天轨
	idx			:INT;			//挡板索引编号
	percent		:REAL;			//比例阀百分比 传入-100~+100
END_VAR
VAR_OUTPUT
END_VAR
VAR
END_VAR

IF percent > 0 THEN
	CASE level OF
		1:
			gController.grd[idx].extendPercent := REAL_TO_WORD(percent * 65535 / 100);
			gController.grd[idx].retractPercent := 0;
		2:
			gController.sky[idx].extendPercent := REAL_TO_WORD(percent * 65535 / 100);
			gController.sky[idx].retractPercent := 0;
	END_CASE
ELSE
	CASE level OF
		1:
			gController.grd[idx].extendPercent := 0;
			gController.grd[idx].retractPercent := REAL_TO_WORD(ABS(percent) * 65535 / 100);
		2:
			gController.sky[idx].extendPercent := 0;
			gController.sky[idx].retractPercent := REAL_TO_WORD(ABS(percent) * 65535 / 100);
	END_CASE
END_IF

END_FUNCTION_BLOCK

// Device/Application/core/pid/grdPosCtrl
FUNCTION_BLOCK grdPosCtrl
VAR_INPUT
	idx			:INT;			//挡板索引编号
	isReset		:BOOL;
	cycTimer	:REAL;
END_VAR
	

VAR_OUTPUT
	res		:REAL;		
END_VAR
VAR
	posPid		:BasePIDCtrl;
	spdPid		:BasePIDCtrl;
	setSpeed	:REAL;
	overBase	:REAL;
	out			:REAL;
	controller	:DevPid;
END_VAR

controller := gDev.grd[idx].ctrl;
posPid(
	Act_Val:= gDev.grd[idx].sensor.position, 
	Set_Val:= controller.pos.Set_Point,
	Kp:= controller.pos.Kp, 
	Ki:= controller.pos.Ki, 
	Kd:= controller.pos.Kd, 
	Y_MAX:= controller.pos.Max_Val,     //最大速度
	Y_MIN:= -controller.pos.Max_Val,    //水平运动正反一致
	rCycle:= 0.1,   //位置计算周期 100ms
	Reset:= isReset, 
	Y => controller.pos.OUT, 
	LimitActive=> );

IF ABS(posPid.Y - setSpeed) > (cycTimer * controller.pos.Max_ACC) THEN
	IF posPid.Y > setSpeed THEN
		setSpeed := setSpeed + (cycTimer * controller.pos.Max_ACC);
	ELSE
		setSpeed := setSpeed - (cycTimer * controller.pos.Max_ACC);
	END_IF
ELSE
	setSpeed := posPid.Y;
END_IF

controller.spd.Set_Point := setSpeed;

IF setSpeed > 0 THEN
	overBase := setSpeed * controller.ff.pstKv + controller.ff.pstThreshold;
ELSE 
	overBase := setSpeed * controller.ff.negKv - controller.ff.negThreshold;
END_IF

spdPid(
	Act_Val:= gDev.grd[idx].sensor.speed, 
	Set_Val:= controller.spd.Set_Point,
	Kp:= controller.spd.Kp, 
	Ki:= controller.spd.Ki, 
	Kd:= controller.spd.Kd, 
	Y_MAX:= controller.spd.Max_Val,     //最大速度
	Y_MIN:= -controller.spd.Max_Val,    //水平运动正反一致
	rCycle:= 0.02,   //位置计算周期 100ms
	Reset:= isReset, 
	Y=> , 
	LimitActive=> );

out := spdPid.Y + overBase;		
IF out > controller.spd.Max_Val THEN
	out := controller.spd.Max_Val;
END_IF
IF out < -controller.spd.Max_Val THEN
	out := -controller.spd.Max_Val;
END_IF
IF isReset	THEN out := 0;	END_IF
controller.spd.OUT := out;
gDev.grd[idx].ctrl := controller;
res := out;

END_FUNCTION_BLOCK

// Device/Application/core/pid/BasePIDCtrl
FUNCTION_BLOCK BasePIDCtrl
VAR_INPUT
	Act_Val 	:REAL;			//实际值
	Set_Val		:REAL;			//设定值
	Kp			:REAL;			
	Ki			:REAL;
	Kd			:REAL;
	Y_MAX		:REAL;
	Y_MIN		:REAL;
	rCycle		:REAL;			//单位/s
	Reset		:BOOL;
END_VAR
VAR_OUTPUT
	Y			:REAL;
	LimitActive	:BOOL;
END_VAR
VAR
	fCycle			:REAL;    
	CycleTime		:TIME ;
	Err				:REAL;    		//本次误差
	LastErr			:REAL;    		//上次误差
	KiErrSum		:REAL;			//积分累计误差
	KdErr			:REAL;			//微分误差
	Result			:REAL;			//计算结果
	Result_OUT		:REAL;		    //限制结果
	trig			:R_TRIG ;
	ton				:TON ;
END_VAR

IF  rCycle < 0.01 THEN  //10ms最小
	fCycle := 0.01;
ELSE
	fCycle := rCycle;
END_IF

CycleTime := REAL_TO_TIME (TIME_TO_REAL(T#1S) * fCycle);
ton (IN := NOT ton.Q ,PT := CycleTime ,Q =>);
trig (CLK := ton.Q  ,Q =>);

IF trig.Q THEN 			//PID计算
	Err := Set_Val - Act_Val;  //误差计算
	KiErrSum := KiErrSum + Err ;   //积分计算
	KdErr := Err -LastErr;    //微分计算
	LastErr := Err;
	(*IF ABS(Err) < 10 THEN		//误差较低时才开启积分
		KiErrSum := KiErrSum + Err ;   //积分计算
	END_IF*)
	Result :=  Kp * Err + Ki * KiErrSum + Kd * KdErr;  
END_IF

IF Result > Y_MAX  THEN         //限幅度输出
	Result_OUT := Y_MAX ;
	LimitActive := TRUE ;
ELSIF Result < Y_MIN THEN
	Result_OUT := Y_MIN  ;
	LimitActive := TRUE ;
ELSE 
	Result_OUT := Result ;
	LimitActive :=FALSE ;
END_IF
IF Reset THEN   //pid 不输出
	KiErrSum := 0;
	KdErr := 0;
	LastErr	:= 0;
	Y := 0;
ELSE
	Y := Result_OUT;	
END_IF

END_FUNCTION_BLOCK

// Device/Application/core/pid/skyPosCtrl
FUNCTION_BLOCK skyPosCtrl
VAR_INPUT
	idx			:INT;			//挡板索引编号
	isReset		:BOOL;
	cycTimer	:REAL;
END_VAR
	

VAR_OUTPUT
	res		:REAL;		
END_VAR
VAR
	posPid		:BasePIDCtrl;
	spdPid		:BasePIDCtrl;
	setSpeed	:REAL;
	overBase	:REAL;
	out			:REAL;
	//fb_Val		:REAL;
	controller	:DevPid;
END_VAR

controller := gDev.sky[idx].ctrl;
posPid(
	Act_Val:= gDev.sky[idx].sensor.position, 
	Set_Val:= controller.pos.Set_Point,
	Kp:= controller.pos.Kp, 
	Ki:= controller.pos.Ki, 
	Kd:= controller.pos.Kd, 
	Y_MAX:= controller.pos.Max_Val,     //最大速度
	Y_MIN:= -controller.pos.Max_Val,    //水平运动正反一致
	rCycle:= 0.05,   //位置计算周期 100ms
	Reset:= isReset, 
	Y => controller.pos.OUT, 
	LimitActive=> );

IF ABS(posPid.Y - setSpeed) > (cycTimer * controller.pos.Max_ACC) THEN
	IF posPid.Y > setSpeed THEN
		setSpeed := setSpeed + (cycTimer * controller.pos.Max_ACC);
	ELSE
		setSpeed := setSpeed - (cycTimer * controller.pos.Max_ACC);
	END_IF
ELSE
	setSpeed := posPid.Y;
END_IF

controller.spd.Set_Point := setSpeed;

IF setSpeed > 0 THEN
	overBase := setSpeed * controller.ff.pstKv + controller.ff.pstThreshold;
END_IF
IF setSpeed < 0 THEN	
	overBase := setSpeed * controller.ff.negKv - controller.ff.negThreshold;
END_IF

spdPid(
	Act_Val:= gDev.sky[idx].sensor.speed, 
	Set_Val:= controller.spd.Set_Point,
	Kp:= controller.spd.Kp, 
	Ki:= controller.spd.Ki, 
	Kd:= controller.spd.Kd, 
	Y_MAX:= controller.spd.Max_Val,     //最大速度
	Y_MIN:= -controller.spd.Max_Val,    //水平运动正反一致
	rCycle:= 0.02,   //位置计算周期 100ms
	Reset:= isReset, 
	Y=> , 
	LimitActive=> );

out := spdPid.Y + overBase;	

	
IF out > controller.spd.Max_Val THEN
	out := controller.spd.Max_Val;
END_IF
IF out < -controller.spd.Max_Val THEN
	out := -controller.spd.Max_Val;
END_IF
IF isReset	THEN out := 0;	END_IF
controller.spd.OUT := out;
gDev.sky[idx].ctrl := controller;
res := out;

END_FUNCTION_BLOCK

// Device/Application/basefun/updateDevStatus
FUNCTION updateDevStatus : DevStatus
VAR_INPUT
	level		:INT;		//1->地轨	2->天轨
	idx			:INT;		//挡板索引编号	
	errorVal	:REAL;		//误差范围
END_VAR
VAR
	extendVal	:REAL;		//伸出值
	retractVal	:REAL;		//缩回到位值
	nowVal		:REAL;		//当前值
	stat		:DevStatus;	//设备状态
END_VAR



(* 本函数用于根据设备的标定伸出/缩回值以及当前位置
** 判断该缸体是否处于伸出/缩回到位状态，如果到位更新参数
*)

stat := DevStatus.unknown;	//初始化状态量
CASE level OF
	1:
		extendVal := gDev.grd[idx].sensor.extendVal;
		retractVal := gDev.grd[idx].sensor.retractVal;
		nowVal := gDev.grd[idx].sensor.position;
		stat := gDev.grd[idx].state;
	2:
		extendVal := gDev.sky[idx].sensor.extendVal;
		retractVal := gDev.sky[idx].sensor.retractVal;
		nowVal := gDev.sky[idx].sensor.position;
		stat := gDev.sky[idx].state;
END_CASE

IF nowVal > 1 THEN
	IF nowVal < retractVal + errorVal THEN
		stat := DevStatus.retracted;
	ELSIF nowVal > extendVal - errorVal THEN
		stat := DevStatus.extended;
	ELSE 
		IF stat <> DevStatus.runing THEN
			stat := DevStatus.error;
		END_IF
	END_IF
ELSE
	stat := DevStatus.unknown;	
END_IF

CASE level OF
	1:
		gDev.grd[idx].state := stat;
	2:
		gDev.sky[idx].state := stat;
END_CASE

updateDevStatus := stat;

END_FUNCTION

// Device/Application/basefun/percentCalc
FUNCTION percentCalc : REAL
VAR_INPUT
	level		:INT;	//1->地轨	2->天轨
	idx			:INT;	//挡板索引编号
END_VAR
VAR
	c			:REAL;
	p			:REAL;
END_VAR


//伸出百分比计算
CASE level OF
	1:
		IF gDev.grd[idx].sensor.position < 3 THEN 
			RETURN;
		END_IF
		c := gDev.grd[idx].sensor.position - gDev.grd[idx].sensor.retractVal;
		p := gDev.grd[idx].sensor.extendVal - gDev.grd[idx].sensor.retractVal;
		percentCalc := c * 100 / p;
	2:
		IF gDev.sky[idx].sensor.position < 3 THEN 
			RETURN;
		END_IF
		c := gDev.sky[idx].sensor.position - gDev.sky[idx].sensor.retractVal;
		p := gDev.sky[idx].sensor.extendVal - gDev.sky[idx].sensor.retractVal;
		percentCalc := c * 100 / p;
END_CASE

END_FUNCTION

// Device/Application/basefun/setButtonByDirect
FUNCTION setButtonByDirect : BOOL
VAR_INPUT
	level		:INT;	//1->地轨	2->天轨
	idx			:INT;	//挡板索引编号
	direct		:TargetDirect;
END_VAR
VAR
END_VAR

//	本函数用于根据输入参数 操作UI界面的按钮变量
CASE level OF
	1:
		IF idx = 0 OR idx > 10 THEN		//参数校验
			RETURN;
		END_IF
		CASE direct OF
			TargetDirect.extend:
				gUI.grd[idx].btnStop := FALSE;
				gUI.grd[idx].btnExtend := TRUE;
				gUI.grd[idx].btnRetract := FALSE;
			TargetDirect.retract:
				gUI.grd[idx].btnStop := FALSE;
				gUI.grd[idx].btnExtend := FALSE;
				gUI.grd[idx].btnRetract := TRUE;
			TargetDirect.stop:
				gUI.grd[idx].btnStop := FALSE;
				gUI.grd[idx].btnExtend := FALSE;
				gUI.grd[idx].btnRetract := FALSE;
		END_CASE
	2:
		IF idx > 10 THEN		//参数校验
			RETURN;
		END_IF
		CASE direct OF
			TargetDirect.extend:
				gUI.sky[idx].btnStop := FALSE;
				gUI.sky[idx].btnExtend := TRUE;
				gUI.sky[idx].btnRetract := FALSE;
			TargetDirect.retract:
				gUI.sky[idx].btnStop := FALSE;
				gUI.sky[idx].btnExtend := FALSE;
				gUI.sky[idx].btnRetract := TRUE;
			TargetDirect.stop:
				gUI.sky[idx].btnStop := FALSE;
				gUI.sky[idx].btnExtend := FALSE;
				gUI.sky[idx].btnRetract := FALSE;
		END_CASE
		
END_CASE

END_FUNCTION

// Device/Application/modbus/ModbusAct
PROGRAM ModbusAct
VAR
	bInit					: BOOL:=TRUE;
	iCountAct				: UINT:=10;	
	connectStatus			: UINT;
	iErrCode				: BYTE;
	idx						: INT;
	logicIdx				: INT;
	gi						: INT;
	si						: INT;		
	iSec					: INT;		//section iterator
	devNum					: WORD;
	fbModbusServer			: ModbusServer;
	inputBuff				: ARRAY[0..1000]OF WORD;
	holdingBuff				: ARRAY[0..1000]OF WORD;
	
	fbModbusClient			: ModbusTcp_Client;
	fbReadHoldRegister  	: ReadHoldRegister;		//读保持寄存器
	fbWriteMutiRegister		: WriteMutiRegister;	
	l2p						: mdbsLogicToPhy;
	p2l						: mdbsPhyToLogic;
	n2i						: mdbsNumToIdx;
	rvs						: DataReverse;
END_VAR

//初始化
IF bInit THEN
	initialize();
	bInit := FALSE;
END_IF

IF connectStatus <> 1 THEN
	fbModbusClient(sIPAddress:='192.168.2.21',uiPort:=520);//连接IPC
	//fbModbusClient(sIPAddress:='192.168.5.55',uiPort:=502);//连接工控机
END_IF

IF fbModbusClient.bSuccess THEN
	connectStatus := 1;	
	CASE iCountAct OF
		10:
			handleCmd();		//接收华中指令
			localCmdHandler();	//处理本机挡板指令 + 启动液压站
		20:
			handleStat1();		//发送状态至华中
		21:
			handleStat2();
		22:
			handleStat3();
	END_CASE
END_IF
		
//做服务器接收天地轨客户端发送的数据
fbModbusServer(	wPort := 512, 
	pInputData := ADR(inputBuff[0]), pOutputData := ADR(holdingBuff[0]), 
	uiInputDataSize := 1000, uiOutputDataSize := 1000, 
	xEnable := TRUE, xReset := FALSE, tTimeout := 1000, 
	xBusy => , xError => , byClientConnections => );


//将缓冲区Buff数据转至本地
localStatHandler();
//updateStat();

ACTION initialize:
gModbus.srv.request.startAddr	:= 10;
gModbus.srv.request.length		:= 48;

gModbus.srv.response.startAddr := 110;
gModbus.srv.response.length := 210;
END_ACTION

METHOD localCmdHandler
VAR_INPUT
END_VAR
VAR
	iBit				:INT;
	exLevel				:INT;
	exIdx				:INT;
	exDirect			:TargetDirect;
	exeDirect			:TargetDirect;

END_VAR
VAR CONSTANT
	no		:ARRAY [1..8] OF INT :=[11, 14, 17, 20, 49, 50, 51, 52];	
END_VAR

FOR iSec := 1 TO 8 DO
	gModbus.srv.request.data[no[iSec]] := gModbus.modbusBuffer[no[iSec]];
END_FOR

FOR iSec := 1 TO 4 DO
	gModbus.srv.request.arrNew[iSec,1	] := gModbus.srv.request.data[no[iSec]].1	;
	gModbus.srv.request.arrNew[iSec,2	] := gModbus.srv.request.data[no[iSec]].2	;
	gModbus.srv.request.arrNew[iSec,3	] := gModbus.srv.request.data[no[iSec]].3	;
	gModbus.srv.request.arrNew[iSec,4	] := gModbus.srv.request.data[no[iSec]].4	;
	gModbus.srv.request.arrNew[iSec,5	] := gModbus.srv.request.data[no[iSec]].5	;
	gModbus.srv.request.arrNew[iSec,6	] := gModbus.srv.request.data[no[iSec]].6	;
	gModbus.srv.request.arrNew[iSec,7	] := gModbus.srv.request.data[no[iSec]].7	;
	gModbus.srv.request.arrNew[iSec,8	] := gModbus.srv.request.data[no[iSec]].8	;
	gModbus.srv.request.arrNew[iSec,9	] := gModbus.srv.request.data[no[iSec]].9	;
	gModbus.srv.request.arrNew[iSec,10	] := gModbus.srv.request.data[no[iSec]].10	;
	gModbus.srv.request.arrNew[iSec,11	] := gModbus.srv.request.data[no[iSec]].11	;
END_FOR
FOR iSec := 1 TO 4 DO
	FOR iBit := 1 TO 11 DO
		IF gModbus.srv.request.arrNew[iSec, iBit] <> gModbus.srv.request.arrLast[iSec, iBit] THEN
			IF gModbus.srv.request.arrNew[iSec, iBit] THEN	//仅执行上升沿
				//specifically output[grd/sky(exLevel), no(exIdx), TargetDirect(exDirect)]
				l2p(section := iSec, lgcIdx := iBit, 
					level => exLevel, phyIdx => exIdx, direct => exDirect);
				exeDirect := rvs.cmdReverse(input := exDirect);		//华中要求伸缩指令及状态翻转
				
				//过滤	机械结构未完成的grd[4] and sky[4]
				IF exIdx = 4 THEN	exeDirect := TargetDirect.stop;	END_IF
				
				setButtonByDirect(level := exLevel, idx := exIdx, direct := exeDirect);
			END_IF
			gModbus.srv.request.arrLast[iSec, iBit] := gModbus.srv.request.arrNew[iSec, iBit];			
		END_IF
	END_FOR
	
END_FOR


devNum := gModbus.modbusBuffer[49];


//新增一键启动液压站

IF gUI.mode.hydPowerOn THEN
	holdingBuff[48] := holdingBuff[48] OR 1;
END_IF
IF gUI.mode.hydPowerOff THEN
	holdingBuff[48] := holdingBuff[48] OR 2;
END_IF
END_METHOD

ACTION updateStat:
(*
//先把天地轨控制器数据同步至本地
FOR idx := 110 TO 319 DO
	gModbus.srv.response.data[idx] := holdingBuff[idx];
END_FOR

//根据实际状态将挡板数据同步至本地
FOR gi := 1 TO 10 DO
	
	//地轨伸出到位检查
	p2l(section := 1, phyIdx := gi, lgcIdx => logicIdx);//logicIdx范围[223,232]
	IF gDev.grd[gi].state = DevStatus.extended THEN
		gModbus.srv.response.data[logicIdx] := 1;
	ELSE
		gModbus.srv.response.data[logicIdx] := 0;
	END_IF
	//地轨缩回到位检查
	p2l(section := 2, phyIdx := gi, lgcIdx => logicIdx);//logicIdx范围[271,280]
	IF gDev.grd[gi].state = DevStatus.retracted THEN
		gModbus.srv.response.data[logicIdx] := 1;
	ELSE
		gModbus.srv.response.data[logicIdx] := 0;
	END_IF
END_FOR

FOR si := 0 TO 10 DO
	//天轨伸出到位检查
	p2l(section := 3, phyIdx := si, lgcIdx => logicIdx);//logicIdx范围[127,137]
	IF gDev.sky[si].state = DevStatus.extended THEN
		gModbus.srv.response.data[logicIdx] := 1;
	ELSE
		gModbus.srv.response.data[logicIdx] := 0;
	END_IF
	//天轨缩回到位检查
	p2l(section := 4, phyIdx := si, lgcIdx => logicIdx);//logicIdx范围[175,185]
	IF gDev.sky[si].state = DevStatus.retracted THEN
		gModbus.srv.response.data[logicIdx] := 1;
	ELSE
		gModbus.srv.response.data[logicIdx] := 0;
	END_IF	
END_FOR
//至此110-309寄存器状态更新完毕，向华中发送时只需在寄存器写入response.data[]数组

IF devNum > 40000 THEN
	n2i(devNo := devNum, level => , idx =>);
	CASE n2i.level OF
		1:
			gModbus.srv.response.data[312] := REAL_TO_WORD(10 * gDev.grd[n2i.idx].sensor.position);
			gModbus.srv.response.data[313] := REAL_TO_WORD(10 * gDev.grd[n2i.idx].sensor.extendVal);
			gModbus.srv.response.data[314] := REAL_TO_WORD(10 * gDev.grd[n2i.idx].sensor.retractVal);
		2:
			gModbus.srv.response.data[312] := REAL_TO_WORD(10 * gDev.sky[n2i.idx].sensor.position);
			gModbus.srv.response.data[313] := REAL_TO_WORD(10 * gDev.sky[n2i.idx].sensor.extendVal);
			gModbus.srv.response.data[314] := REAL_TO_WORD(10 * gDev.sky[n2i.idx].sensor.retractVal);
	END_CASE
END_IF
*)
END_ACTION

ACTION handleCmd:
fbReadHoldRegister(
	xExecute	:= TRUE,
	slaveId		:= 1,
	wStartAdr	:= gModbus.srv.request.startAddr,
	wLen		:= gModbus.srv.request.length,
	pTcpStream	:= fbModbusClient.pfbTcpStream,
	modbusHoldRegData:= gModbus.modbusBuffer);
	

IF fbReadHoldRegister.bSucced THEN
	fbReadHoldRegister(xExecute := FALSE,
						modbusHoldRegData:=g_modbusHoldRegData);

	//使用holdingBuff接收供给链控制指令，在下一轮循环中作为服务器保持该数据
	FOR idx := 10 TO 57 DO			//startAddr to startAddr+length-1
		holdingBuff[idx] := gModbus.modbusBuffer[idx];
	END_FOR
	
	iCountAct := 20;		
END_IF

IF fbReadHoldRegister.berror THEN
	fbReadHoldRegister(xExecute :=FALSE,
						modbusHoldRegData:= gModbus.modbusBuffer);
	fbModbusClient.M_Reset();
	connectStatus := 0;
	iCountAct := 10;	
	iErrCode := fbReadHoldRegister.errCode;
END_IF
END_ACTION

ACTION handleStat1:


fbWriteMutiRegister(
	xExecute	:= TRUE,
	slaveId		:= 1,
	startAddr	:= 110, //gModbus.srv.response.startAddr 110-319
	wRegNum		:= 70,
	value		:= ADR(gModbus.srv.response.data[110]),
	pTcpStream	:= fbModbusClient.pfbTcpStream);
	
IF fbWriteMutiRegister.bSucced THEN
	fbWriteMutiRegister(xExecute := FALSE);
	iCountAct:= 21;
END_IF

IF fbWriteMutiRegister.berror THEN
	fbWriteMutiRegister(xExecute := FALSE);
	fbModbusClient.M_Reset();
	iCountAct := 10;
	connectStatus := 0;
	iErrCode := fbWriteMutiRegister.errCode;
END_IF
END_ACTION

ACTION handleStat2:


fbWriteMutiRegister(
	xExecute	:= TRUE,
	slaveId		:= 1,
	startAddr	:= 180, //gModbus.srv.response.startAddr 110-319
	wRegNum		:= 70,
	value		:= ADR(gModbus.srv.response.data[180]),
	pTcpStream	:= fbModbusClient.pfbTcpStream);
	
IF fbWriteMutiRegister.bSucced THEN
	fbWriteMutiRegister(xExecute := FALSE);
	iCountAct:= 22;
END_IF

IF fbWriteMutiRegister.berror THEN
	fbWriteMutiRegister(xExecute := FALSE);
	fbModbusClient.M_Reset();
	iCountAct := 10;
	connectStatus := 0;
	iErrCode := fbWriteMutiRegister.errCode;
END_IF
END_ACTION

ACTION handleStat3:


fbWriteMutiRegister(
	xExecute	:= TRUE,
	slaveId		:= 1,
	startAddr	:= 250, //gModbus.srv.response.startAddr 110-319
	wRegNum		:= 70,
	value		:= ADR(gModbus.srv.response.data[250]),
	pTcpStream	:= fbModbusClient.pfbTcpStream);
	
IF fbWriteMutiRegister.bSucced THEN
	fbWriteMutiRegister(xExecute := FALSE);
	iCountAct:= 10;
END_IF

IF fbWriteMutiRegister.berror THEN
	fbWriteMutiRegister(xExecute := FALSE);
	fbModbusClient.M_Reset();
	iCountAct := 10;
	connectStatus := 0;
	iErrCode := fbWriteMutiRegister.errCode;
END_IF
END_ACTION

METHOD localStatHandler : TargetDirect
VAR_INPUT
END_VAR

//先把天地轨控制器数据同步至本地
FOR idx := 110 TO 319 DO
	gModbus.srv.response.data[idx] := holdingBuff[idx];
END_FOR

//根据实际状态将挡板数据同步至本地
FOR gi := 1 TO 10 DO
	(*******************************
	伸缩反向判定，伸出到位返回缩回到位
	**********************************)
	
	//地轨伸出到位检查
	p2l(section := 1, phyIdx := gi, lgcIdx => logicIdx);//logicIdx范围[223,232]
	IF gDev.grd[gi].state = DevStatus.retracted THEN
		gModbus.srv.response.data[logicIdx] := 1;
	ELSE
		gModbus.srv.response.data[logicIdx] := 0;
	END_IF
	//地轨缩回到位检查
	p2l(section := 2, phyIdx := gi, lgcIdx => logicIdx);//logicIdx范围[271,280]
	IF gDev.grd[gi].state = DevStatus.extended THEN
		gModbus.srv.response.data[logicIdx] := 1;
	ELSE
		gModbus.srv.response.data[logicIdx] := 0;
	END_IF
END_FOR

FOR si := 0 TO 10 DO
	//天轨伸出到位检查
	p2l(section := 3, phyIdx := si, lgcIdx => logicIdx);//logicIdx范围[127,137]
	
	
	IF gDev.sky[si].state = DevStatus.retracted THEN
		gModbus.srv.response.data[logicIdx] := 1;
	ELSE
		gModbus.srv.response.data[logicIdx] := 0;
	END_IF
	//天轨缩回到位检查
	p2l(section := 4, phyIdx := si, lgcIdx => logicIdx);//logicIdx范围[175,185]
	IF gDev.sky[si].state = DevStatus.extended THEN
		gModbus.srv.response.data[logicIdx] := 1;
	ELSE
		gModbus.srv.response.data[logicIdx] := 0;
	END_IF	
END_FOR
//至此110-309寄存器状态更新完毕，向华中发送时只需在寄存器写入response.data[]数组

IF devNum > 40000 THEN
	n2i(devNo := devNum, level => , idx =>);
	CASE n2i.level OF
		1:
			gModbus.srv.response.data[312] := REAL_TO_WORD(10 * gDev.grd[n2i.idx].sensor.position);
			gModbus.srv.response.data[313] := REAL_TO_WORD(10 * gDev.grd[n2i.idx].sensor.extendVal);
			gModbus.srv.response.data[314] := REAL_TO_WORD(10 * gDev.grd[n2i.idx].sensor.retractVal);
		2:
			gModbus.srv.response.data[312] := REAL_TO_WORD(10 * gDev.sky[n2i.idx].sensor.position);
			gModbus.srv.response.data[313] := REAL_TO_WORD(10 * gDev.sky[n2i.idx].sensor.extendVal);
			gModbus.srv.response.data[314] := REAL_TO_WORD(10 * gDev.sky[n2i.idx].sensor.retractVal);
	END_CASE
END_IF
END_METHOD

END_PROGRAM

// Device/Application/modbus/mdbsLogicToPhy
FUNCTION_BLOCK mdbsLogicToPhy	//modbus华中挡板地址编号对应本地索引编号
VAR_INPUT
	section		:INT;	//区域限定(1:skyExt, 2:skyRet, 3:grdExt, 4:grdRet)
	lgcIdx		:INT;	//华中对应的地址	10,14{1..10}  17,20{1..11}
END_VAR
VAR_OUTPUT
	level		:INT;	//1->地轨	2->天轨
	phyIdx		:INT;	//内存物理地址对应数组索引
	direct		:TargetDirect;
END_VAR
VAR
END_VAR

(**
 * 将华中指令解析为要动作挡板的标号
 * (level:1->地轨	2->天轨)(phyIdx:内存物理地址对应数组索引)
 *)
CASE section OF
	1://区域限定(1:skyExtend)
		level := 2;
		direct := TargetDirect.extend;
		CASE lgcIdx OF
			1:	phyIdx := 1;		//横1	->	sky1
			2:	phyIdx := 3;		//横2	->	sky3
			3:	phyIdx := 4;		//横3	->	sky4
			4:	phyIdx := 5;		//横4	->	sky5
			5:	phyIdx := 6;		//横5	->	sky6
			6:	phyIdx := 8;		//横6	->	sky8
			7:	phyIdx := 9;		//横7	->	sky9
			8:	phyIdx := 10;		//横8	->	sky10
			9:	phyIdx := 2;		//纵1	->	sky2
			10:	phyIdx := 7;		//纵2	->	sky7
			11:	phyIdx := 0;		//起竖	->	sky0
		END_CASE

	2://区域限定(2:skyRetract)
		level := 2;
		direct := TargetDirect.retract;
		CASE lgcIdx OF
			1:	phyIdx := 1;		//横1	->	sky1
			2:	phyIdx := 3;		//横2	->	sky3
			3:	phyIdx := 4;		//横3	->	sky4
			4:	phyIdx := 5;		//横4	->	sky5
			5:	phyIdx := 6;		//横5	->	sky6
			6:	phyIdx := 8;		//横6	->	sky8
			7:	phyIdx := 9;		//横7	->	sky9
			8:	phyIdx := 10;		//横8	->	sky10
			9:	phyIdx := 2;		//纵1	->	sky2
			10:	phyIdx := 7;		//纵2	->	sky7
			11:	phyIdx := 0;		//起竖	->	sky0
		END_CASE

	3://区域限定(3:grdExtend)
		level := 1;
		direct := TargetDirect.extend;
		CASE lgcIdx OF
			1:	phyIdx := 1;		//横1	->	grd1
			2:	phyIdx := 3;		//横2	->	grd3
			3:	phyIdx := 4;		//横3	->	grd4
			4:	phyIdx := 5;		//横4	->	grd5
			5:	phyIdx := 6;		//横5	->	grd6
			6:	phyIdx := 8;		//横6	->	grd8
			7:	phyIdx := 9;		//横7	->	grd9
			8:	phyIdx := 10;		//横8	->	grd10
			9:	phyIdx := 2;		//纵1	->	grd2
			10:	phyIdx := 7;		//纵2	->	grd7
		END_CASE
	4://区域限定(4:grdRetract)
		level := 1;
		direct := TargetDirect.retract;
		CASE lgcIdx OF
			1:	phyIdx := 1;
			2:	phyIdx := 3;
			3:	phyIdx := 4;
			4:	phyIdx := 5;
			5:	phyIdx := 6;
			6:	phyIdx := 8;
			7:	phyIdx := 9;
			8:	phyIdx := 10;
			9:	phyIdx := 2;
			10:	phyIdx := 7;
		END_CASE
END_CASE

END_FUNCTION_BLOCK

// Device/Application/modbus/mdbsPhyToLogic
FUNCTION_BLOCK mdbsPhyToLogic	//modbus本地索引对应回传华中的状态地址
VAR_INPUT
	section		:INT;	//区域限定(1:grdExt, 2:grdRet, 3:skyExt, 4:skyRet)
	phyIdx		:INT;	//内存物理地址对应数组索引
END_VAR
VAR_OUTPUT
	lgcIdx		:INT;	//华中对应的地址	127 175 223 271...
END_VAR
VAR
END_VAR

(**
 * 输入挡板标号，返回华中需要的寄存器地址号
 *)
CASE section OF
	1://区域限定(1:groundExtend)
		CASE phyIdx OF
			1:	lgcIdx := 223;		//grd1e	->	横1	223
			2:	lgcIdx := 231;		//grd2e	->	纵1	231
			3:	lgcIdx := 224;		//grd3e	->	横2	224
			4:	lgcIdx := 225;		//grd4e	->	横3	225
			5:	lgcIdx := 226;		//grd5e	->	横4	226
			6:	lgcIdx := 227;		//grd6e	->	横5	227
			7:	lgcIdx := 232;		//grd7e	->	纵2	232
			8:	lgcIdx := 228;		//grd8e	->	横6	228
			9:	lgcIdx := 229;		//grd9e	->	横7	229
			10:	lgcIdx := 230;		//grd10e->	横8	230
		END_CASE
	2://区域限定(2:groundRetract)
		CASE phyIdx OF
			1:	lgcIdx := 271;		//grd1r	->	横1
			2:	lgcIdx := 279;		//grd2r	->	纵1
			3:	lgcIdx := 272;		//grd3r	->	横2
			4:	lgcIdx := 273;		//grd4r	->	横3
			5:	lgcIdx := 274;		//grd5r	->	横4
			6:	lgcIdx := 275;		//grd6r	->	横5
			7:	lgcIdx := 280;		//grd7r	->	纵2
			8:	lgcIdx := 276;		//grd8r	->	横6
			9:	lgcIdx := 277;		//grd9r	->	横7
			10:	lgcIdx := 278;		//grd10r->	横8
		END_CASE
	3://区域限定(3:skyExtend)
		CASE phyIdx OF
			0:	lgcIdx := 137;		//sky0e	->	起竖	
			1:	lgcIdx := 127;		//sky1e	->	横1	
			2:	lgcIdx := 135;		//sky2e	->	纵1	
			3:	lgcIdx := 128;		//sky3e	->	横2	
			4:	lgcIdx := 129;		//sky4e	->	横3	
			5:	lgcIdx := 130;		//sky5e	->	横4	
			6:	lgcIdx := 131;		//sky6e	->	横5	
			7:	lgcIdx := 136;		//sky7e	->	纵2	
			8:	lgcIdx := 132;		//sky8e	->	横6	
			9:	lgcIdx := 133;		//sky9e	->	横7	
			10:	lgcIdx := 134;		//sky10e->	横8	
		END_CASE
	
